LIN {X 0,Y 467.921,Z 515.715,A -85,B 0,C 180,E1 -7661.262,E2 -7661.262} C_VEL
LIN {X 0,Y 468.367,Z 505.748,A -85,B 0,C 180,E1 -7662.288,E2 -7662.288} C_VEL
LIN {X 0,Y 468.874,Z 494.586,A -85,B 0,C 180,E1 -7663.217,E2 -7663.217} C_VEL
LIN {X 0,Y 469.352,Z 483.029,A -85,B 0,C 180,E1 -7663.975,E2 -7663.975} C_VEL
LIN {X 0,Y 469.873,Z 469.859,A -85,B 0,C 180,E1 -7664.623,E2 -7664.623} C_VEL
LIN {X 0,Y 468.217,Z 456.623,A -85,B 0,C 180,E1 -7665.144,E2 -7665.144} C_VEL
LIN {X 0,Y 467.024,Z 448.323,A -85,B 0,C 180,E1 -7665.389,E2 -7665.389} C_VEL
LIN {X 0,Y 467.272,Z 438.89,A -85,B 0,C 180,E1 -7668.638,E2 -7668.638} C_VEL
LIN {X 0,Y 467.516,Z 429.097,A -85,B 0,C 180,E1 -7672.077,E2 -7672.077} C_VEL
LIN {X 0,Y 467.845,Z 420.214,A -85,B 0,C 180,E1 -7675.278,E2 -7675.278} C_VEL
LIN {X 0,Y 468.188,Z 412.234,A -85,B 0,C 180,E1 -7678.222,E2 -7678.222} C_VEL
LIN {X 0,Y 468.623,Z 404.282,A -85,B 0,C 180,E1 -7681.258,E2 -7681.258} C_VEL
LIN {X 0,Y 469.224,Z 395.561,A -85,B 0,C 180,E1 -7684.694,E2 -7684.694} C_VEL
LIN {X 0,Y 469.214,Z 392.362,A -85,B 0,C 180,E1 -7686.018,E2 -7686.018} C_VEL
LIN {X 0,Y 468.571,Z 387.882,A -85,B 0,C 180,E1 -7687.951,E2 -7687.951} C_VEL
LIN {X 0,Y 467.585,Z 382.244,A -85,B 0,C 180,E1 -7690.549,E2 -7690.549} C_VEL
LIN {X 0,Y 467.557,Z 382.244,A -85,B 0,C 180,E1 -7693.82,E2 -7693.82} C_VEL
LIN {X 0,Y 467.559,Z 382.245,A -85,B 0,C 180,E1 -7696.255,E2 -7696.255} C_VEL
LIN {X 0,Y 467.579,Z 382.244,A -85,B 0,C 180,E1 -7698.726,E2 -7698.726} C_VEL
LIN {X 0,Y 467.573,Z 382.242,A -85,B 0,C 180,E1 -7701.956,E2 -7701.956} C_VEL
LIN {X 0,Y 467.568,Z 382.246,A -85,B 0,C 180,E1 -7705.167,E2 -7705.167} C_VEL
LIN {X 0,Y 467.591,Z 382.241,A -85,B 0,C 180,E1 -7708.26,E2 -7708.26} C_VEL
LIN {X 0,Y 467.566,Z 382.244,A -85,B 0,C 180,E1 -7711.249,E2 -7711.249} C_VEL
LIN {X 0,Y 467.581,Z 382.24,A -85,B 0,C 180,E1 -7714.158,E2 -7714.158} C_VEL
LIN {X 0,Y 467.588,Z 382.242,A -85,B 0,C 180,E1 -7716.996,E2 -7716.996} C_VEL
LIN {X 0,Y 467.634,Z 382.236,A -85,B 0,C 180,E1 -7719.777,E2 -7719.777} C_VEL
LIN {X 0,Y 467.609,Z 382.238,A -85,B 0,C 180,E1 -7722.506,E2 -7722.506} C_VEL
LIN {X 0,Y 467.61,Z 382.24,A -85,B 0,C 180,E1 -7725.196,E2 -7725.196} C_VEL
LIN {X 0,Y 467.667,Z 382.231,A -85,B 0,C 180,E1 -7727.854,E2 -7727.854} C_VEL
LIN {X 0,Y 467.679,Z 382.23,A -85,B 0,C 180,E1 -7731.356,E2 -7731.356} C_VEL
LIN {X 0,Y 467.736,Z 382.221,A -85,B 0,C 180,E1 -7733.962,E2 -7733.962} C_VEL
LIN {X 0,Y 467.866,Z 382.208,A -85,B 0,C 180,E1 -7737.416,E2 -7737.416} C_VEL
LIN {X 0,Y 467.889,Z 382.203,A -85,B 0,C 180,E1 -7739.999,E2 -7739.999} C_VEL
LIN {X 0,Y 467.857,Z 382.208,A -85,B 0,C 180,E1 -7742.582,E2 -7742.582} C_VEL
LIN {X 0,Y 467.72,Z 382.224,A -85,B 0,C 180,E1 -7746.037,E2 -7746.037} C_VEL
LIN {X 0,Y 467.672,Z 382.231,A -85,B 0,C 180,E1 -7748.642,E2 -7748.642} C_VEL
LIN {X 0,Y 467.665,Z 382.232,A -85,B 0,C 180,E1 -7752.144,E2 -7752.144} C_VEL
LIN {X 0,Y 467.647,Z 382.232,A -85,B 0,C 180,E1 -7755.694,E2 -7755.694} C_VEL
LIN {X 0,Y 467.629,Z 382.235,A -85,B 0,C 180,E1 -7759.307,E2 -7759.307} C_VEL
LIN {X 0,Y 467.542,Z 382.247,A -85,B 0,C 180,E1 -7762.073,E2 -7762.073} C_VEL
LIN {X 0,Y 467.592,Z 382.241,A -85,B 0,C 180,E1 -7764.887,E2 -7764.887} C_VEL
LIN {X 0,Y 467.616,Z 382.235,A -85,B 0,C 180,E1 -7767.768,E2 -7767.768} C_VEL
LIN {X 0,Y 467.574,Z 382.244,A -85,B 0,C 180,E1 -7771.043,E2 -7771.043} C_VEL
LIN {X 0,Y 467.594,Z 382.241,A -85,B 0,C 180,E1 -7774.24,E2 -7774.24} C_VEL
LIN {X 0,Y 467.548,Z 382.246,A -85,B 0,C 180,E1 -7777.183,E2 -7777.183} C_VEL
LIN {X 0,Y 467.575,Z 382.244,A -85,B 0,C 180,E1 -7780.264,E2 -7780.264} C_VEL
LIN {X 0,Y 467.565,Z 382.244,A -85,B 0,C 180,E1 -7782.561,E2 -7782.561} C_VEL
LIN {X 0,Y 467.569,Z 382.243,A -85,B 0,C 180,E1 -7785.05,E2 -7785.05} C_VEL
LIN {X 0,Y 467.577,Z 382.244,A -85,B 0,C 180,E1 -7788.595,E2 -7788.595} C_VEL
LIN {X 0,Y 467.569,Z 382.243,A -85,B 0,C 180,E1 -7791.953,E2 -7791.953} C_VEL
LIN {X 0,Y 467.57,Z 382.243,A -85,B 0,C 180,E1 -7795.165,E2 -7795.165} C_VEL
LIN {X 0,Y 467.585,Z 382.242,A -85,B 0,C 180,E1 -7798.257,E2 -7798.257} C_VEL
LIN {X 0,Y 467.576,Z 382.241,A -85,B 0,C 180,E1 -7801.248,E2 -7801.248} C_VEL
LIN {X 0,Y 467.611,Z 382.239,A -85,B 0,C 180,E1 -7804.158,E2 -7804.158} C_VEL
LIN {X 0,Y 467.577,Z 382.243,A -85,B 0,C 180,E1 -7806.993,E2 -7806.993} C_VEL
LIN {X 0,Y 467.622,Z 382.237,A -85,B 0,C 180,E1 -7809.774,E2 -7809.774} C_VEL
LIN {X 0,Y 467.605,Z 382.242,A -85,B 0,C 180,E1 -7812.504,E2 -7812.504} C_VEL
LIN {X 0,Y 467.595,Z 382.239,A -85,B 0,C 180,E1 -7815.401,E2 -7815.401} C_VEL
LIN {X 0,Y 466.923,Z 382.325,A -85,B 0,C 180,E1 -7816.12,E2 -7816.12} C_VEL
LIN {X 0,Y 464.081,Z 382.675,A -85,B 0,C 180,E1 -7817.288,E2 -7817.288} C_VEL
LIN {X 0,Y 461.683,Z 382.978,A -85,B 0,C 180,E1 -7818.23,E2 -7818.23} C_VEL
LIN {X 0,Y 460.656,Z 383.105,A -85,B 0,C 180,E1 -7818.958,E2 -7818.958} C_VEL
LIN {X 0,Y 460.574,Z 383.113,A -85,B 0,C 180,E1 -7819.205,E2 -7819.205} C_VEL
LIN {X 0,Y 460.711,Z 383.098,A -85,B 0,C 180,E1 -7822.539,E2 -7822.539} C_VEL
LIN {X 0,Y 460.689,Z 383.1,A -85,B 0,C 180,E1 -7824.745,E2 -7824.745} C_VEL
LIN {X 0,Y 460.794,Z 383.087,A -85,B 0,C 180,E1 -7827.374,E2 -7827.374} C_VEL
LIN {X 0,Y 460.845,Z 383.083,A -85,B 0,C 180,E1 -7829.997,E2 -7829.997} C_VEL
LIN {X 0,Y 460.816,Z 383.086,A -85,B 0,C 180,E1 -7832.619,E2 -7832.619} C_VEL
LIN {X 0,Y 460.702,Z 383.099,A -85,B 0,C 180,E1 -7836.127,E2 -7836.127} C_VEL
LIN {X 0,Y 460.618,Z 383.109,A -85,B 0,C 180,E1 -7838.773,E2 -7838.773} C_VEL
LIN {X 0,Y 460.621,Z 383.109,A -85,B 0,C 180,E1 -7842.453,E2 -7842.453} C_VEL
LIN {X 0,Y 460.606,Z 383.113,A -85,B 0,C 180,E1 -7846.004,E2 -7846.004} C_VEL
LIN {X 0,Y 460.552,Z 383.117,A -85,B 0,C 180,E1 -7849.612,E2 -7849.612} C_VEL
LIN {X 0,Y 460.497,Z 383.126,A -85,B 0,C 180,E1 -7852.425,E2 -7852.425} C_VEL
LIN {X 0,Y 460.526,Z 383.12,A -85,B 0,C 180,E1 -7855.292,E2 -7855.292} C_VEL
LIN {X 0,Y 460.314,Z 383.15,A -85,B 0,C 180,E1 -7858.244,E2 -7858.244} C_VEL
LIN {X 0,Y 459.937,Z 383.378,A -85,B 0,C 180,E1 -7861.296,E2 -7861.296} C_VEL
LIN {X 0,Y 459.851,Z 386.637,A -85,B 0,C 180,E1 -7864.43,E2 -7864.43} C_VEL
LIN {X 0,Y 459.799,Z 390.069,A -85,B 0,C 180,E1 -7867.685,E2 -7867.685} C_VEL
LIN {X 0,Y 459.766,Z 392.69,A -85,B 0,C 180,E1 -7870.157,E2 -7870.157} C_VEL
LIN {X 0,Y 459.691,Z 396.273,A -85,B 0,C 180,E1 -7873.464,E2 -7873.464} C_VEL
LIN {X 0,Y 459.701,Z 399.614,A -85,B 0,C 180,E1 -7876.494,E2 -7876.494} C_VEL
LIN {X 0,Y 463.013,Z 414.025,A -85,B 0,C 180,E1 -7877.08,E2 -7877.08} C_VEL
LIN {X 0,Y 463.229,Z 419.464,A -85,B 0,C 180,E1 -7877.321,E2 -7877.321} C_VEL
LIN {X 0,Y 462.847,Z 431.199,A -85,B 0,C 180,E1 -7877.934,E2 -7877.934} C_VEL
LIN {X 0,Y 462.335,Z 443.116,A -85,B 0,C 180,E1 -7878.751,E2 -7878.751} C_VEL
LIN {X 0,Y 461.772,Z 454.579,A -85,B 0,C 180,E1 -7879.747,E2 -7879.747} C_VEL
LIN {X 0,Y 461.288,Z 464.913,A -85,B 0,C 180,E1 -7880.883,E2 -7880.883} C_VEL
LIN {X 0,Y 460.796,Z 474.093,A -85,B 0,C 180,E1 -7882.13,E2 -7882.13} C_VEL
LIN {X 0,Y 460.424,Z 482.007,A -85,B 0,C 180,E1 -7883.467,E2 -7883.467} C_VEL
LIN {X 0,Y 460.136,Z 488.259,A -85,B 0,C 180,E1 -7884.791,E2 -7884.791} C_VEL
LIN {X 0,Y 459.903,Z 493.202,A -85,B 0,C 180,E1 -7886.104,E2 -7886.104} C_VEL
LIN {X 0,Y 459.764,Z 497.612,A -85,B 0,C 180,E1 -7887.656,E2 -7887.656} C_VEL
LIN {X 0,Y 459.612,Z 500.119,A -85,B 0,C 180,E1 -7888.895,E2 -7888.895} C_VEL
LIN {X 0,Y 459.544,Z 502.273,A -85,B 0,C 180,E1 -7890.65,E2 -7890.65} C_VEL
LIN {X 0,Y 459.507,Z 502.75,A -85,B 0,C 180,E1 -7891.698,E2 -7891.698} C_VEL
LIN {X 0,Y 459.506,Z 502.726,A -85,B 0,C 180,E1 -7892.689,E2 -7892.689} C_VEL
LIN {X 0,Y 459.591,Z 501.374,A -85,B 0,C 180,E1 -7894.44,E2 -7894.44} C_VEL
LIN {X 0,Y 459.697,Z 499.578,A -85,B 0,C 180,E1 -7895.621,E2 -7895.621} C_VEL
LIN {X 0,Y 459.851,Z 496.301,A -85,B 0,C 180,E1 -7897.064,E2 -7897.064} C_VEL
LIN {X 0,Y 460.043,Z 491.012,A -85,B 0,C 180,E1 -7898.717,E2 -7898.717} C_VEL
LIN {X 0,Y 460.329,Z 484.96,A -85,B 0,C 180,E1 -7900.142,E2 -7900.142} C_VEL
LIN {X 0,Y 460.726,Z 477.332,A -85,B 0,C 180,E1 -7901.548,E2 -7901.548} C_VEL
LIN {X 0,Y 461.138,Z 469.536,A -85,B 0,C 180,E1 -7902.712,E2 -7902.712} C_VEL
LIN {X 0,Y 461.631,Z 459.665,A -85,B 0,C 180,E1 -7903.913,E2 -7903.913} C_VEL
LIN {X 0,Y 462.141,Z 449.461,A -85,B 0,C 180,E1 -7904.905,E2 -7904.905} C_VEL
LIN {X 0,Y 462.714,Z 437.651,A -85,B 0,C 180,E1 -7905.824,E2 -7905.824} C_VEL
LIN {X 0,Y 463.137,Z 426.76,A -85,B 0,C 180,E1 -7906.488,E2 -7906.488} C_VEL
LIN {X 0,Y 463.465,Z 416.28,A -85,B 0,C 180,E1 -7906.981,E2 -7906.981} C_VEL
LIN {X 0,Y 460.771,Z 404.535,A -85,B 0,C 180,E1 -7907.495,E2 -7907.495} C_VEL
LIN {X 0,Y 459.906,Z 400.872,A -85,B 0,C 180,E1 -7907.648,E2 -7907.648} C_VEL
LIN {X 0,Y 459.915,Z 397.286,A -85,B 0,C 180,E1 -7911.211,E2 -7911.211} C_VEL
LIN {X 0,Y 460.001,Z 394.662,A -85,B 0,C 180,E1 -7913.861,E2 -7913.861} C_VEL
LIN {X 0,Y 460.164,Z 392.942,A -85,B 0,C 180,E1 -7915.621,E2 -7915.621} C_VEL
LIN {X 0,Y 460.271,Z 389.556,A -85,B 0,C 180,E1 -7919.126,E2 -7919.126} C_VEL
LIN {X 0,Y 460.513,Z 387.881,A -85,B 0,C 180,E1 -7920.875,E2 -7920.875} C_VEL
LIN {X 0,Y 460.546,Z 383.831,A -85,B 0,C 180,E1 -7925.254,E2 -7925.254} C_VEL
LIN {X 0,Y 460.524,Z 383.125,A -85,B 0,C 180,E1 -7926.133,E2 -7926.133} C_VEL
LIN {X 0,Y 460.593,Z 383.116,A -85,B 0,C 180,E1 -7927.894,E2 -7927.894} C_VEL
LIN {X 0,Y 460.584,Z 383.116,A -85,B 0,C 180,E1 -7930.551,E2 -7930.551} C_VEL
LIN {X 0,Y 460.559,Z 383.119,A -85,B 0,C 180,E1 -7933.233,E2 -7933.233} C_VEL
LIN {X 0,Y 460.586,Z 383.114,A -85,B 0,C 180,E1 -7936.009,E2 -7936.009} C_VEL
LIN {X 0,Y 460.542,Z 383.12,A -85,B 0,C 180,E1 -7938.906,E2 -7938.906} C_VEL
LIN {X 0,Y 460.531,Z 383.119,A -85,B 0,C 180,E1 -7941.486,E2 -7941.486} C_VEL
LIN {X 0,Y 460.523,Z 383.119,A -85,B 0,C 180,E1 -7944.334,E2 -7944.334} C_VEL
LIN {X 0,Y 460.553,Z 383.117,A -85,B 0,C 180,E1 -7947.246,E2 -7947.246} C_VEL
LIN {X 0,Y 460.497,Z 383.124,A -85,B 0,C 180,E1 -7950.242,E2 -7950.242} C_VEL
LIN {X 0,Y 460.501,Z 383.124,A -85,B 0,C 180,E1 -7953.328,E2 -7953.328} C_VEL
LIN {X 0,Y 460.455,Z 383.13,A -85,B 0,C 180,E1 -7956.532,E2 -7956.532} C_VEL
LIN {X 0,Y 460.56,Z 383.118,A -85,B 0,C 180,E1 -7959.86,E2 -7959.86} C_VEL
LIN {X 0,Y 460.52,Z 383.125,A -85,B 0,C 180,E1 -7962.908,E2 -7962.908} C_VEL
LIN {X 0,Y 460.502,Z 383.126,A -85,B 0,C 180,E1 -7965.832,E2 -7965.832} C_VEL
LIN {X 0,Y 460.554,Z 383.166,A -85,B 0,C 180,E1 -7968.151,E2 -7968.151} C_VEL
LIN {X 0,Y 461.514,Z 388.734,A -85,B 0,C 180,E1 -7971.371,E2 -7971.371} C_VEL
LIN {X 0,Y 462.217,Z 393.26,A -85,B 0,C 180,E1 -7973.695,E2 -7973.695} C_VEL
LIN {X 0,Y 462.049,Z 397.702,A -85,B 0,C 180,E1 -7975.756,E2 -7975.756} C_VEL
LIN {X 0,Y 461.476,Z 404.849,A -85,B 0,C 180,E1 -7978.82,E2 -7978.82} C_VEL
LIN {X 0,Y 460.949,Z 413.207,A -85,B 0,C 180,E1 -7982.168,E2 -7982.168} C_VEL
LIN {X 0,Y 460.688,Z 419.887,A -85,B 0,C 180,E1 -7984.717,E2 -7984.717} C_VEL
LIN {X 0,Y 460.362,Z 428.911,A -85,B 0,C 180,E1 -7988.04,E2 -7988.04} C_VEL
LIN {X 0,Y 460.132,Z 436.905,A -85,B 0,C 180,E1 -7990.879,E2 -7990.879} C_VEL
LIN {X 0,Y 459.921,Z 446.946,A -85,B 0,C 180,E1 -7994.338,E2 -7994.338} C_VEL
LIN {X 0,Y 461.798,Z 460.563,A -85,B 0,C 180,E1 -7994.778,E2 -7994.778} C_VEL
LIN {X 0,Y 462.902,Z 471.743,A -85,B 0,C 180,E1 -7995.271,E2 -7995.271} C_VEL
LIN {X 0,Y 462.342,Z 483.982,A -85,B 0,C 180,E1 -7995.927,E2 -7995.927} C_VEL
LIN {X 0,Y 461.725,Z 496.525,A -85,B 0,C 180,E1 -7996.806,E2 -7996.806} C_VEL
LIN {X 0,Y 461.226,Z 506.53,A -85,B 0,C 180,E1 -7997.686,E2 -7997.686} C_VEL
LIN {X 0,Y 460.792,Z 516.676,A -85,B 0,C 180,E1 -7998.79,E2 -7998.79} C_VEL
LIN {X 0,Y 460.32,Z 526.54,A -85,B 0,C 180,E1 -8000.113,E2 -8000.113} C_VEL
LIN {X 0,Y 460.02,Z 534.432,A -85,B 0,C 180,E1 -8001.437,E2 -8001.437} C_VEL
LIN {X 0,Y 459.773,Z 541.699,A -85,B 0,C 180,E1 -8002.979,E2 -8002.979} C_VEL
LIN {X 0,Y 459.681,Z 546.549,A -85,B 0,C 180,E1 -8004.3,E2 -8004.3} C_VEL
LIN {X 0,Y 459.58,Z 550.258,A -85,B 0,C 180,E1 -8005.618,E2 -8005.618} C_VEL
LIN {X 0,Y 459.626,Z 552.182,A -85,B 0,C 180,E1 -8006.497,E2 -8006.497} C_VEL
LIN {X 0,Y 459.621,Z 553.624,A -85,B 0,C 180,E1 -8007.374,E2 -8007.374} C_VEL
LIN {X 0,Y 459.63,Z 554.658,A -85,B 0,C 180,E1 -8008.251,E2 -8008.251} C_VEL
LIN {X 0,Y 459.554,Z 555.294,A -85,B 0,C 180,E1 -8009.127,E2 -8009.127} C_VEL
LIN {X 0,Y 459.531,Z 555.527,A -85,B 0,C 180,E1 -8010.003,E2 -8010.003} C_VEL
LIN {X 0,Y 459.631,Z 554.72,A -85,B 0,C 180,E1 -8011.756,E2 -8011.756} C_VEL
LIN {X 0,Y 459.623,Z 553.72,A -85,B 0,C 180,E1 -8012.632,E2 -8012.632} C_VEL
LIN {X 0,Y 459.627,Z 552.303,A -85,B 0,C 180,E1 -8013.51,E2 -8013.51} C_VEL
LIN {X 0,Y 459.63,Z 549.329,A -85,B 0,C 180,E1 -8014.827,E2 -8014.827} C_VEL
LIN {X 0,Y 459.719,Z 544.241,A -85,B 0,C 180,E1 -8016.434,E2 -8016.434} C_VEL
LIN {X 0,Y 459.896,Z 538.06,A -85,B 0,C 180,E1 -8017.908,E2 -8017.908} C_VEL
LIN {X 0,Y 460.18,Z 531.048,A -85,B 0,C 180,E1 -8019.231,E2 -8019.231} C_VEL
LIN {X 0,Y 460.527,Z 522.257,A -85,B 0,C 180,E1 -8020.555,E2 -8020.555} C_VEL
LIN {X 0,Y 461.13,Z 512.301,A -85,B 0,C 180,E1 -8021.765,E2 -8021.765} C_VEL
LIN {X 0,Y 461.487,Z 502.127,A -85,B 0,C 180,E1 -8022.765,E2 -8022.765} C_VEL
LIN {X 0,Y 462.02,Z 491.009,A -85,B 0,C 180,E1 -8023.64,E2 -8023.64} C_VEL
LIN {X 0,Y 462.655,Z 478.556,A -85,B 0,C 180,E1 -8024.406,E2 -8024.406} C_VEL
LIN {X 0,Y 462.896,Z 469.283,A -85,B 0,C 180,E1 -8024.848,E2 -8024.848} C_VEL
LIN {X 0,Y 461.122,Z 455.923,A -85,B 0,C 180,E1 -8025.384,E2 -8025.384} C_VEL
LIN {X 0,Y 459.94,Z 447.939,A -85,B 0,C 180,E1 -8025.636,E2 -8025.636} C_VEL
LIN {X 0,Y 460.202,Z 439.025,A -85,B 0,C 180,E1 -8028.765,E2 -8028.765} C_VEL
LIN {X 0,Y 460.426,Z 430.104,A -85,B 0,C 180,E1 -8031.963,E2 -8031.963} C_VEL
LIN {X 0,Y 460.747,Z 422.328,A -85,B 0,C 180,E1 -8034.804,E2 -8034.804} C_VEL
LIN {X 0,Y 461.158,Z 413.292,A -85,B 0,C 180,E1 -8038.195,E2 -8038.195} C_VEL
LIN {X 0,Y 461.579,Z 405.572,A -85,B 0,C 180,E1 -8041.18,E2 -8041.18} C_VEL
LIN {X 0,Y 462.254,Z 396.524,A -85,B 0,C 180,E1 -8044.814,E2 -8044.814} C_VEL
LIN {X 0,Y 462.171,Z 392.819,A -85,B 0,C 180,E1 -8046.377,E2 -8046.377} C_VEL
LIN {X 0,Y 461.232,Z 386.951,A -85,B 0,C 180,E1 -8049.003,E2 -8049.003} C_VEL
LIN {X 0,Y 460.557,Z 383.119,A -85,B 0,C 180,E1 -8050.813,E2 -8050.813} C_VEL
LIN {X 0,Y 460.517,Z 383.121,A -85,B 0,C 180,E1 -8054.17,E2 -8054.17} C_VEL
LIN {X 0,Y 460.493,Z 383.126,A -85,B 0,C 180,E1 -8057.105,E2 -8057.105} C_VEL
LIN {X 0,Y 460.526,Z 383.12,A -85,B 0,C 180,E1 -8060.136,E2 -8060.136} C_VEL
LIN {X 0,Y 460.485,Z 383.127,A -85,B 0,C 180,E1 -8063.471,E2 -8063.471} C_VEL
LIN {X 0,Y 460.529,Z 383.121,A -85,B 0,C 180,E1 -8066.674,E2 -8066.674} C_VEL
LIN {X 0,Y 460.52,Z 383.12,A -85,B 0,C 180,E1 -8069.76,E2 -8069.76} C_VEL
LIN {X 0,Y 460.542,Z 383.119,A -85,B 0,C 180,E1 -8072.754,E2 -8072.754} C_VEL
LIN {X 0,Y 460.535,Z 383.121,A -85,B 0,C 180,E1 -8075.667,E2 -8075.667} C_VEL
LIN {X 0,Y 460.535,Z 383.119,A -85,B 0,C 180,E1 -8078.578,E2 -8078.578} C_VEL
LIN {X 0,Y 460.598,Z 383.114,A -85,B 0,C 180,E1 -8081.311,E2 -8081.311} C_VEL
LIN {X 0,Y 460.618,Z 383.109,A -85,B 0,C 180,E1 -8084.059,E2 -8084.059} C_VEL
LIN {X 0,Y 460.621,Z 383.109,A -85,B 0,C 180,E1 -8087.665,E2 -8087.665} C_VEL
LIN {X 0,Y 460.629,Z 383.108,A -85,B 0,C 180,E1 -8091.223,E2 -8091.223} C_VEL
LIN {X 0,Y 460.703,Z 383.097,A -85,B 0,C 180,E1 -8093.869,E2 -8093.869} C_VEL
LIN {X 0,Y 460.807,Z 383.087,A -85,B 0,C 180,E1 -8097.377,E2 -8097.377} C_VEL
LIN {X 0,Y 460.859,Z 383.079,A -85,B 0,C 180,E1 -8099.999,E2 -8099.999} C_VEL
LIN {X 0,Y 460.798,Z 383.088,A -85,B 0,C 180,E1 -8102.622,E2 -8102.622} C_VEL
LIN {X 0,Y 460.684,Z 383.1,A -85,B 0,C 180,E1 -8106.129,E2 -8106.129} C_VEL
LIN {X 0,Y 460.623,Z 383.109,A -85,B 0,C 180,E1 -8108.775,E2 -8108.775} C_VEL
LIN {X 0,Y 460.606,Z 383.113,A -85,B 0,C 180,E1 -8112.434,E2 -8112.434} C_VEL
LIN {X 0,Y 460.61,Z 383.109,A -85,B 0,C 180,E1 -8115.996,E2 -8115.996} C_VEL
LIN {X 0,Y 460.576,Z 383.113,A -85,B 0,C 180,E1 -8119.614,E2 -8119.614} C_VEL
LIN {X 0,Y 460.518,Z 383.122,A -85,B 0,C 180,E1 -8122.427,E2 -8122.427} C_VEL
LIN {X 0,Y 460.556,Z 383.117,A -85,B 0,C 180,E1 -8125.795,E2 -8125.795} C_VEL
LIN {X 0,Y 460.546,Z 383.118,A -85,B 0,C 180,E1 -8128.232,E2 -8128.232} C_VEL
LIN {X 0,Y 460.527,Z 383.119,A -85,B 0,C 180,E1 -8131.281,E2 -8131.281} C_VEL
LIN {X 0,Y 460.537,Z 383.12,A -85,B 0,C 180,E1 -8134.503,E2 -8134.503} C_VEL
LIN {X 0,Y 460.504,Z 383.123,A -85,B 0,C 180,E1 -8137.622,E2 -8137.622} C_VEL
LIN {X 0,Y 460.539,Z 383.12,A -85,B 0,C 180,E1 -8140.266,E2 -8140.266} C_VEL
LIN {X 0,Y 460.513,Z 383.121,A -85,B 0,C 180,E1 -8143.372,E2 -8143.372} C_VEL
LIN {X 0,Y 460.513,Z 383.123,A -85,B 0,C 180,E1 -8146.623,E2 -8146.623} C_VEL
LIN {X 0,Y 460.538,Z 383.119,A -85,B 0,C 180,E1 -8149.73,E2 -8149.73} C_VEL
LIN {X 0,Y 460.504,Z 383.126,A -85,B 0,C 180,E1 -8152.522,E2 -8152.522} C_VEL
LIN {X 0,Y 460.551,Z 383.117,A -85,B 0,C 180,E1 -8155.622,E2 -8155.622} C_VEL
LIN {X 0,Y 460.54,Z 383.12,A -85,B 0,C 180,E1 -8158.742,E2 -8158.742} C_VEL
LIN {X 0,Y 460.582,Z 383.115,A -85,B 0,C 180,E1 -8162.252,E2 -8162.252} C_VEL
LIN {X 0,Y 460.56,Z 383.117,A -85,B 0,C 180,E1 -8164.703,E2 -8164.703} C_VEL
LIN {X 0,Y 460.511,Z 383.123,A -85,B 0,C 180,E1 -8167.569,E2 -8167.569} C_VEL
LIN {X 0,Y 460.568,Z 383.116,A -85,B 0,C 180,E1 -8170.382,E2 -8170.382} C_VEL
LIN {X 0,Y 460.562,Z 383.114,A -85,B 0,C 180,E1 -8173.143,E2 -8173.143} C_VEL
LIN {X 0,Y 460.552,Z 383.118,A -85,B 0,C 180,E1 -8175.865,E2 -8175.865} C_VEL
LIN {X 0,Y 460.608,Z 383.111,A -85,B 0,C 180,E1 -8178.556,E2 -8178.556} C_VEL
LIN {X 0,Y 460.574,Z 383.113,A -85,B 0,C 180,E1 -8179.205,E2 -8179.205} C_VEL
LIN {X 0,Y 459.917,Z 383.198,A -85,B 0,C 180,E1 -8179.935,E2 -8179.935} C_VEL
LIN {X 0,Y 457.097,Z 383.552,A -85,B 0,C 180,E1 -8181.121,E2 -8181.121} C_VEL
LIN {X 0,Y 454.716,Z 383.847,A -85,B 0,C 180,E1 -8182.078,E2 -8182.078} C_VEL
LIN {X 0,Y 453.703,Z 383.971,A -85,B 0,C 180,E1 -8182.817,E2 -8182.817} C_VEL
LIN {X 0,Y 453.625,Z 383.98,A -85,B 0,C 180,E1 -8183.067,E2 -8183.067} C_VEL
LIN {X 0,Y 453.663,Z 383.976,A -85,B 0,C 180,E1 -8184.664,E2 -8184.664} C_VEL
LIN {X 0,Y 453.738,Z 383.966,A -85,B 0,C 180,E1 -8187.333,E2 -8187.333} C_VEL
LIN {X 0,Y 453.815,Z 383.959,A -85,B 0,C 180,E1 -8189.997,E2 -8189.997} C_VEL
LIN {X 0,Y 453.756,Z 383.964,A -85,B 0,C 180,E1 -8192.66,E2 -8192.66} C_VEL
LIN {X 0,Y 453.669,Z 383.976,A -85,B 0,C 180,E1 -8196.222,E2 -8196.222} C_VEL
LIN {X 0,Y 453.582,Z 383.985,A -85,B 0,C 180,E1 -8198.91,E2 -8198.91} C_VEL
LIN {X 0,Y 453.588,Z 383.984,A -85,B 0,C 180,E1 -8202.547,E2 -8202.547} C_VEL
LIN {X 0,Y 453.541,Z 383.992,A -85,B 0,C 180,E1 -8206.192,E2 -8206.192} C_VEL
LIN {X 0,Y 453.504,Z 383.995,A -85,B 0,C 180,E1 -8209.038,E2 -8209.038} C_VEL
LIN {X 0,Y 453.46,Z 384.002,A -85,B 0,C 180,E1 -8211.833,E2 -8211.833} C_VEL
LIN {X 0,Y 453.49,Z 383.995,A -85,B 0,C 180,E1 -8214.731,E2 -8214.731} C_VEL
LIN {X 0,Y 453.337,Z 384.018,A -85,B 0,C 180,E1 -8217.711,E2 -8217.711} C_VEL
LIN {X 0,Y 452.926,Z 384.075,A -85,B 0,C 180,E1 -8220.796,E2 -8220.796} C_VEL
LIN {X 0,Y 452.874,Z 384.19,A -85,B 0,C 180,E1 -8221.405,E2 -8221.405} C_VEL
LIN {X 0,Y 452.794,Z 387.534,A -85,B 0,C 180,E1 -8224.652,E2 -8224.652} C_VEL
LIN {X 0,Y 452.747,Z 390.692,A -85,B 0,C 180,E1 -8227.66,E2 -8227.66} C_VEL
LIN {X 0,Y 452.681,Z 393.925,A -85,B 0,C 180,E1 -8230.691,E2 -8230.691} C_VEL
LIN {X 0,Y 452.634,Z 397.827,A -85,B 0,C 180,E1 -8234.317,E2 -8234.317} C_VEL
LIN {X 0,Y 452.641,Z 399.971,A -85,B 0,C 180,E1 -8236.268,E2 -8236.268} C_VEL
LIN {X 0,Y 455.934,Z 414.289,A -85,B 0,C 180,E1 -8236.852,E2 -8236.852} C_VEL
LIN {X 0,Y 456.407,Z 418.655,A -85,B 0,C 180,E1 -8237.057,E2 -8237.057} C_VEL
LIN {X 0,Y 455.989,Z 431.188,A -85,B 0,C 180,E1 -8237.708,E2 -8237.708} C_VEL
LIN {X 0,Y 455.444,Z 443.242,A -85,B 0,C 180,E1 -8238.541,E2 -8238.541} C_VEL
LIN {X 0,Y 454.832,Z 454.602,A -85,B 0,C 180,E1 -8239.537,E2 -8239.537} C_VEL
LIN {X 0,Y 454.359,Z 464.73,A -85,B 0,C 180,E1 -8240.653,E2 -8240.653} C_VEL
LIN {X 0,Y 453.789,Z 474.492,A -85,B 0,C 180,E1 -8241.99,E2 -8241.99} C_VEL
LIN {X 0,Y 453.402,Z 482.206,A -85,B 0,C 180,E1 -8243.307,E2 -8243.307} C_VEL
LIN {X 0,Y 453.091,Z 488.725,A -85,B 0,C 180,E1 -8244.706,E2 -8244.706} C_VEL
LIN {X 0,Y 452.848,Z 493.644,A -85,B 0,C 180,E1 -8246.035,E2 -8246.035} C_VEL
LIN {X 0,Y 452.704,Z 498.061,A -85,B 0,C 180,E1 -8247.617,E2 -8247.617} C_VEL
LIN {X 0,Y 452.505,Z 501.043,A -85,B 0,C 180,E1 -8249.168,E2 -8249.168} C_VEL
LIN {X 0,Y 452.468,Z 502.495,A -85,B 0,C 180,E1 -8250.428,E2 -8250.428} C_VEL
LIN {X 0,Y 452.416,Z 503.013,A -85,B 0,C 180,E1 -8251.213,E2 -8251.213} C_VEL
LIN {X 0,Y 452.411,Z 503.197,A -85,B 0,C 180,E1 -8252.299,E2 -8252.299} C_VEL
LIN {X 0,Y 452.446,Z 502.892,A -85,B 0,C 180,E1 -8253.227,E2 -8253.227} C_VEL
LIN {X 0,Y 452.504,Z 502.069,A -85,B 0,C 180,E1 -8254.254,E2 -8254.254} C_VEL
LIN {X 0,Y 452.55,Z 500.783,A -85,B 0,C 180,E1 -8255.21,E2 -8255.21} C_VEL
LIN {X 0,Y 452.745,Z 497.722,A -85,B 0,C 180,E1 -8256.752,E2 -8256.752} C_VEL
LIN {X 0,Y 452.914,Z 493.826,A -85,B 0,C 180,E1 -8258.136,E2 -8258.136} C_VEL
LIN {X 0,Y 453.151,Z 488.507,A -85,B 0,C 180,E1 -8259.577,E2 -8259.577} C_VEL
LIN {X 0,Y 453.485,Z 481.699,A -85,B 0,C 180,E1 -8261.008,E2 -8261.008} C_VEL
LIN {X 0,Y 453.982,Z 473.16,A -85,B 0,C 180,E1 -8262.431,E2 -8262.431} C_VEL
LIN {X 0,Y 454.522,Z 464.332,A -85,B 0,C 180,E1 -8263.613,E2 -8263.613} C_VEL
LIN {X 0,Y 454.983,Z 454.695,A -85,B 0,C 180,E1 -8264.662,E2 -8264.662} C_VEL
LIN {X 0,Y 455.57,Z 444.076,A -85,B 0,C 180,E1 -8265.597,E2 -8265.597} C_VEL
LIN {X 0,Y 456.09,Z 432.537,A -85,B 0,C 180,E1 -8266.407,E2 -8266.407} C_VEL
LIN {X 0,Y 456.573,Z 419.658,A -85,B 0,C 180,E1 -8267.087,E2 -8267.087} C_VEL
LIN {X 0,Y 456.28,Z 415.433,A -85,B 0,C 180,E1 -8267.284,E2 -8267.284} C_VEL
LIN {X 0,Y 452.856,Z 401.356,A -85,B 0,C 180,E1 -8267.903,E2 -8267.903} C_VEL
LIN {X 0,Y 452.864,Z 398.185,A -85,B 0,C 180,E1 -8271.073,E2 -8271.073} C_VEL
LIN {X 0,Y 452.95,Z 395.562,A -85,B 0,C 180,E1 -8273.766,E2 -8273.766} C_VEL
LIN {X 0,Y 453.126,Z 393.81,A -85,B 0,C 180,E1 -8275.553,E2 -8275.553} C_VEL
LIN {X 0,Y 453.227,Z 390.435,A -85,B 0,C 180,E1 -8279.112,E2 -8279.112} C_VEL
LIN {X 0,Y 453.478,Z 388.773,A -85,B 0,C 180,E1 -8280.889,E2 -8280.889} C_VEL
LIN {X 0,Y 453.522,Z 384.723,A -85,B 0,C 180,E1 -8285.336,E2 -8285.336} C_VEL
LIN {X 0,Y 453.482,Z 384.003,A -85,B 0,C 180,E1 -8286.229,E2 -8286.229} C_VEL
LIN {X 0,Y 453.541,Z 383.994,A -85,B 0,C 180,E1 -8288.017,E2 -8288.017} C_VEL
LIN {X 0,Y 453.535,Z 383.993,A -85,B 0,C 180,E1 -8290.717,E2 -8290.717} C_VEL
LIN {X 0,Y 453.504,Z 383.998,A -85,B 0,C 180,E1 -8293.442,E2 -8293.442} C_VEL
LIN {X 0,Y 453.523,Z 383.996,A -85,B 0,C 180,E1 -8296.197,E2 -8296.197} C_VEL
LIN {X 0,Y 453.491,Z 383.999,A -85,B 0,C 180,E1 -8299.045,E2 -8299.045} C_VEL
LIN {X 0,Y 453.472,Z 383.999,A -85,B 0,C 180,E1 -8301.837,E2 -8301.837} C_VEL
LIN {X 0,Y 453.498,Z 383.995,A -85,B 0,C 180,E1 -8304.736,E2 -8304.736} C_VEL
LIN {X 0,Y 453.508,Z 383.995,A -85,B 0,C 180,E1 -8307.964,E2 -8307.964} C_VEL
LIN {X 0,Y 453.454,Z 384.002,A -85,B 0,C 180,E1 -8310.762,E2 -8310.762} C_VEL
LIN {X 0,Y 453.45,Z 384.003,A -85,B 0,C 180,E1 -8313.916,E2 -8313.916} C_VEL
LIN {X 0,Y 453.447,Z 384.003,A -85,B 0,C 180,E1 -8317.191,E2 -8317.191} C_VEL
LIN {X 0,Y 453.512,Z 383.996,A -85,B 0,C 180,E1 -8319.448,E2 -8319.448} C_VEL
LIN {X 0,Y 453.469,Z 384.003,A -85,B 0,C 180,E1 -8322.995,E2 -8322.995} C_VEL
LIN {X 0,Y 453.455,Z 384.003,A -85,B 0,C 180,E1 -8325.784,E2 -8325.784} C_VEL
LIN {X 0,Y 453.512,Z 384.041,A -85,B 0,C 180,E1 -8327.718,E2 -8327.718} C_VEL
LIN {X 0,Y 454.354,Z 388.949,A -85,B 0,C 180,E1 -8330.662,E2 -8330.662} C_VEL
LIN {X 0,Y 455.183,Z 394.03,A -85,B 0,C 180,E1 -8333.407,E2 -8333.407} C_VEL
LIN {X 0,Y 455.156,Z 397.71,A -85,B 0,C 180,E1 -8335.163,E2 -8335.163} C_VEL
LIN {X 0,Y 454.571,Z 404.727,A -85,B 0,C 180,E1 -8338.292,E2 -8338.292} C_VEL
LIN {X 0,Y 453.923,Z 413.613,A -85,B 0,C 180,E1 -8341.949,E2 -8341.949} C_VEL
LIN {X 0,Y 453.634,Z 420.872,A -85,B 0,C 180,E1 -8344.787,E2 -8344.787} C_VEL
LIN {X 0,Y 453.275,Z 429.888,A -85,B 0,C 180,E1 -8348.158,E2 -8348.158} C_VEL
LIN {X 0,Y 453.045,Z 438.125,A -85,B 0,C 180,E1 -8351.136,E2 -8351.136} C_VEL
LIN {X 0,Y 452.853,Z 446.636,A -85,B 0,C 180,E1 -8354.078,E2 -8354.078} C_VEL
LIN {X 0,Y 454.775,Z 459.997,A -85,B 0,C 180,E1 -8354.525,E2 -8354.525} C_VEL
LIN {X 0,Y 455.963,Z 472.582,A -85,B 0,C 180,E1 -8355.099,E2 -8355.099} C_VEL
LIN {X 0,Y 455.333,Z 485.389,A -85,B 0,C 180,E1 -8355.82,E2 -8355.82} C_VEL
LIN {X 0,Y 454.801,Z 496.155,A -85,B 0,C 180,E1 -8356.601,E2 -8356.601} C_VEL
LIN {X 0,Y 454.245,Z 506.142,A -85,B 0,C 180,E1 -8357.494,E2 -8357.494} C_VEL
LIN {X 0,Y 453.792,Z 516.278,A -85,B 0,C 180,E1 -8358.615,E2 -8358.615} C_VEL
LIN {X 0,Y 453.268,Z 526.122,A -85,B 0,C 180,E1 -8359.958,E2 -8359.958} C_VEL
LIN {X 0,Y 452.952,Z 534.004,A -85,B 0,C 180,E1 -8361.302,E2 -8361.302} C_VEL
LIN {X 0,Y 452.693,Z 541.267,A -85,B 0,C 180,E1 -8362.869,E2 -8362.869} C_VEL
LIN {X 0,Y 452.579,Z 546.123,A -85,B 0,C 180,E1 -8364.21,E2 -8364.21} C_VEL
LIN {X 0,Y 452.501,Z 549.841,A -85,B 0,C 180,E1 -8365.549,E2 -8365.549} C_VEL
LIN {X 0,Y 452.525,Z 551.766,A -85,B 0,C 180,E1 -8366.442,E2 -8366.442} C_VEL
LIN {X 0,Y 452.543,Z 553.212,A -85,B 0,C 180,E1 -8367.333,E2 -8367.333} C_VEL
LIN {X 0,Y 452.538,Z 554.25,A -85,B 0,C 180,E1 -8368.223,E2 -8368.223} C_VEL
LIN {X 0,Y 452.49,Z 554.888,A -85,B 0,C 180,E1 -8369.113,E2 -8369.113} C_VEL
LIN {X 0,Y 452.465,Z 555.121,A -85,B 0,C 180,E1 -8370.003,E2 -8370.003} C_VEL
LIN {X 0,Y 452.49,Z 554.913,A -85,B 0,C 180,E1 -8370.893,E2 -8370.893} C_VEL
LIN {X 0,Y 452.539,Z 554.311,A -85,B 0,C 180,E1 -8371.783,E2 -8371.783} C_VEL
LIN {X 0,Y 452.545,Z 553.311,A -85,B 0,C 180,E1 -8372.674,E2 -8372.674} C_VEL
LIN {X 0,Y 452.526,Z 551.888,A -85,B 0,C 180,E1 -8373.565,E2 -8373.565} C_VEL
LIN {X 0,Y 452.561,Z 548.911,A -85,B 0,C 180,E1 -8374.903,E2 -8374.903} C_VEL
LIN {X 0,Y 452.615,Z 544.309,A -85,B 0,C 180,E1 -8376.399,E2 -8376.399} C_VEL
LIN {X 0,Y 452.843,Z 537.624,A -85,B 0,C 180,E1 -8378.032,E2 -8378.032} C_VEL
LIN {X 0,Y 453.116,Z 530.596,A -85,B 0,C 180,E1 -8379.376,E2 -8379.376} C_VEL
LIN {X 0,Y 453.514,Z 521.793,A -85,B 0,C 180,E1 -8380.72,E2 -8380.72} C_VEL
LIN {X 0,Y 454.117,Z 511.821,A -85,B 0,C 180,E1 -8381.949,E2 -8381.949} C_VEL
LIN {X 0,Y 454.497,Z 501.621,A -85,B 0,C 180,E1 -8382.965,E2 -8382.965} C_VEL
LIN {X 0,Y 455.075,Z 490.489,A -85,B 0,C 180,E1 -8383.853,E2 -8383.853} C_VEL
LIN {X 0,Y 455.778,Z 478.015,A -85,B 0,C 180,E1 -8384.628,E2 -8384.628} C_VEL
LIN {X 0,Y 455.93,Z 469.98,A -85,B 0,C 180,E1 -8385.023,E2 -8385.023} C_VEL
LIN {X 0,Y 454.204,Z 456.5,A -85,B 0,C 180,E1 -8385.585,E2 -8385.585} C_VEL
LIN {X 0,Y 452.896,Z 447.599,A -85,B 0,C 180,E1 -8385.875,E2 -8385.875} C_VEL
LIN {X 0,Y 453.121,Z 438.857,A -85,B 0,C 180,E1 -8389.012,E2 -8389.012} C_VEL
LIN {X 0,Y 453.4,Z 429.781,A -85,B 0,C 180,E1 -8392.322,E2 -8392.322} C_VEL
LIN {X 0,Y 453.736,Z 422.048,A -85,B 0,C 180,E1 -8395.214,E2 -8395.214} C_VEL
LIN {X 0,Y 454.186,Z 413.034,A -85,B 0,C 180,E1 -8398.668,E2 -8398.668} C_VEL
LIN {X 0,Y 454.655,Z 405.211,A -85,B 0,C 180,E1 -8401.768,E2 -8401.768} C_VEL
LIN {X 0,Y 455.241,Z 397.682,A -85,B 0,C 180,E1 -8404.837,E2 -8404.837} C_VEL
LIN {X 0,Y 455.131,Z 393.64,A -85,B 0,C 180,E1 -8406.585,E2 -8406.585} C_VEL
LIN {X 0,Y 453.93,Z 386.239,A -85,B 0,C 180,E1 -8409.983,E2 -8409.983} C_VEL
LIN {X 0,Y 453.501,Z 383.998,A -85,B 0,C 180,E1 -8411.124,E2 -8411.124} C_VEL
LIN {X 0,Y 453.494,Z 383.997,A -85,B 0,C 180,E1 -8414.529,E2 -8414.529} C_VEL
LIN {X 0,Y 453.462,Z 384,A -85,B 0,C 180,E1 -8418.07,E2 -8418.07} C_VEL
LIN {X 0,Y 453.46,Z 384.001,A -85,B 0,C 180,E1 -8420.802,E2 -8420.802} C_VEL
LIN {X 0,Y 453.463,Z 384,A -85,B 0,C 180,E1 -8423.917,E2 -8423.917} C_VEL
LIN {X 0,Y 453.487,Z 383.998,A -85,B 0,C 180,E1 -8427.151,E2 -8427.151} C_VEL
LIN {X 0,Y 453.479,Z 383.997,A -85,B 0,C 180,E1 -8430.268,E2 -8430.268} C_VEL
LIN {X 0,Y 453.476,Z 384.001,A -85,B 0,C 180,E1 -8433.291,E2 -8433.291} C_VEL
LIN {X 0,Y 453.506,Z 383.995,A -85,B 0,C 180,E1 -8436.238,E2 -8436.238} C_VEL
LIN {X 0,Y 453.495,Z 383.997,A -85,B 0,C 180,E1 -8439.118,E2 -8439.118} C_VEL
LIN {X 0,Y 453.515,Z 383.992,A -85,B 0,C 180,E1 -8441.944,E2 -8441.944} C_VEL
LIN {X 0,Y 453.548,Z 383.99,A -85,B 0,C 180,E1 -8444.726,E2 -8444.726} C_VEL
LIN {X 0,Y 453.568,Z 383.988,A -85,B 0,C 180,E1 -8448.378,E2 -8448.378} C_VEL
LIN {X 0,Y 453.595,Z 383.985,A -85,B 0,C 180,E1 -8451.086,E2 -8451.086} C_VEL
LIN {X 0,Y 453.67,Z 383.973,A -85,B 0,C 180,E1 -8453.774,E2 -8453.774} C_VEL
LIN {X 0,Y 453.751,Z 383.966,A -85,B 0,C 180,E1 -8457.336,E2 -8457.336} C_VEL
LIN {X 0,Y 453.829,Z 383.954,A -85,B 0,C 180,E1 -8459.999,E2 -8459.999} C_VEL
LIN {X 0,Y 453.742,Z 383.967,A -85,B 0,C 180,E1 -8462.663,E2 -8462.663} C_VEL
LIN {X 0,Y 453.651,Z 383.976,A -85,B 0,C 180,E1 -8466.225,E2 -8466.225} C_VEL
LIN {X 0,Y 453.59,Z 383.985,A -85,B 0,C 180,E1 -8468.913,E2 -8468.913} C_VEL
LIN {X 0,Y 453.574,Z 383.988,A -85,B 0,C 180,E1 -8472.528,E2 -8472.528} C_VEL
LIN {X 0,Y 453.554,Z 383.989,A -85,B 0,C 180,E1 -8476.195,E2 -8476.195} C_VEL
LIN {X 0,Y 453.526,Z 383.993,A -85,B 0,C 180,E1 -8479.038,E2 -8479.038} C_VEL
LIN {X 0,Y 453.485,Z 383.997,A -85,B 0,C 180,E1 -8481.835,E2 -8481.835} C_VEL
LIN {X 0,Y 453.507,Z 383.996,A -85,B 0,C 180,E1 -8484.734,E2 -8484.734} C_VEL
LIN {X 0,Y 453.531,Z 383.99,A -85,B 0,C 180,E1 -8487.956,E2 -8487.956} C_VEL
LIN {X 0,Y 453.472,Z 383.997,A -85,B 0,C 180,E1 -8491.523,E2 -8491.523} C_VEL
LIN {X 0,Y 453.493,Z 383.999,A -85,B 0,C 180,E1 -8494.775,E2 -8494.775} C_VEL
LIN {X 0,Y 453.463,Z 384.001,A -85,B 0,C 180,E1 -8498.31,E2 -8498.31} C_VEL
LIN {X 0,Y 453.499,Z 383.998,A -85,B 0,C 180,E1 -8500.607,E2 -8500.607} C_VEL
LIN {X 0,Y 453.464,Z 384.001,A -85,B 0,C 180,E1 -8504.22,E2 -8504.22} C_VEL
LIN {X 0,Y 453.453,Z 384.003,A -85,B 0,C 180,E1 -8507.001,E2 -8507.001} C_VEL
LIN {X 0,Y 453.498,Z 383.995,A -85,B 0,C 180,E1 -8509.407,E2 -8509.407} C_VEL
LIN {X 0,Y 453.456,Z 384.001,A -85,B 0,C 180,E1 -8512.808,E2 -8512.808} C_VEL
LIN {X 0,Y 453.481,Z 383.998,A -85,B 0,C 180,E1 -8516.085,E2 -8516.085} C_VEL
LIN {X 0,Y 453.478,Z 383.998,A -85,B 0,C 180,E1 -8519.238,E2 -8519.238} C_VEL
LIN {X 0,Y 453.537,Z 383.992,A -85,B 0,C 180,E1 -8522.295,E2 -8522.295} C_VEL
LIN {X 0,Y 453.515,Z 383.992,A -85,B 0,C 180,E1 -8525.263,E2 -8525.263} C_VEL
LIN {X 0,Y 453.48,Z 384.001,A -85,B 0,C 180,E1 -8528.412,E2 -8528.412} C_VEL
LIN {X 0,Y 453.521,Z 383.994,A -85,B 0,C 180,E1 -8531.006,E2 -8531.006} C_VEL
LIN {X 0,Y 453.567,Z 383.988,A -85,B 0,C 180,E1 -8533.877,E2 -8533.877} C_VEL
LIN {X 0,Y 453.561,Z 383.986,A -85,B 0,C 180,E1 -8537.468,E2 -8537.468} C_VEL
LIN {X 0,Y 453.588,Z 383.983,A -85,B 0,C 180,E1 -8541.084,E2 -8541.084} C_VEL
LIN {X 0,Y 453.625,Z 383.98,A -85,B 0,C 180,E1 -8543.067,E2 -8543.067} C_VEL
LIN {X 0,Y 452.939,Z 384.066,A -85,B 0,C 180,E1 -8543.808,E2 -8543.808} C_VEL
LIN {X 0,Y 449.992,Z 384.431,A -85,B 0,C 180,E1 -8545.01,E2 -8545.01} C_VEL
LIN {X 0,Y 447.567,Z 384.737,A -85,B 0,C 180,E1 -8545.979,E2 -8545.979} C_VEL
LIN {X 0,Y 446.623,Z 384.853,A -85,B 0,C 180,E1 -8546.729,E2 -8546.729} C_VEL
LIN {X 0,Y 446.598,Z 384.854,A -85,B 0,C 180,E1 -8546.983,E2 -8546.983} C_VEL
LIN {X 0,Y 446.785,Z 384.834,A -85,B 0,C 180,E1 -8549.997,E2 -8549.997} C_VEL
LIN {X 0,Y 446.7,Z 384.843,A -85,B 0,C 180,E1 -8552.702,E2 -8552.702} C_VEL
LIN {X 0,Y 446.638,Z 384.852,A -85,B 0,C 180,E1 -8556.32,E2 -8556.32} C_VEL
LIN {X 0,Y 446.528,Z 384.863,A -85,B 0,C 180,E1 -8559.052,E2 -8559.052} C_VEL
LIN {X 0,Y 446.52,Z 384.864,A -85,B 0,C 180,E1 -8562.726,E2 -8562.726} C_VEL
LIN {X 0,Y 446.48,Z 384.87,A -85,B 0,C 180,E1 -8566.455,E2 -8566.455} C_VEL
LIN {X 0,Y 446.452,Z 384.873,A -85,B 0,C 180,E1 -8569.3,E2 -8569.3} C_VEL
LIN {X 0,Y 446.402,Z 384.881,A -85,B 0,C 180,E1 -8572.196,E2 -8572.196} C_VEL
LIN {X 0,Y 446.427,Z 384.875,A -85,B 0,C 180,E1 -8575.15,E2 -8575.15} C_VEL
LIN {X 0,Y 446.233,Z 384.904,A -85,B 0,C 180,E1 -8578.191,E2 -8578.191} C_VEL
LIN {X 0,Y 445.842,Z 384.957,A -85,B 0,C 180,E1 -8581.34,E2 -8581.34} C_VEL
LIN {X 0,Y 445.734,Z 388.154,A -85,B 0,C 180,E1 -8584.579,E2 -8584.579} C_VEL
LIN {X 0,Y 445.651,Z 391.667,A -85,B 0,C 180,E1 -8587.955,E2 -8587.955} C_VEL
LIN {X 0,Y 445.625,Z 394.677,A -85,B 0,C 180,E1 -8590.8,E2 -8590.8} C_VEL
LIN {X 0,Y 445.538,Z 398.064,A -85,B 0,C 180,E1 -8593.946,E2 -8593.946} C_VEL
LIN {X 0,Y 445.599,Z 400.514,A -85,B 0,C 180,E1 -8596.04,E2 -8596.04} C_VEL
LIN {X 0,Y 448.792,Z 414.199,A -85,B 0,C 180,E1 -8596.605,E2 -8596.605} C_VEL
LIN {X 0,Y 449.545,Z 419.114,A -85,B 0,C 180,E1 -8596.845,E2 -8596.845} C_VEL
LIN {X 0,Y 449.094,Z 431.724,A -85,B 0,C 180,E1 -8597.513,E2 -8597.513} C_VEL
LIN {X 0,Y 448.589,Z 442.428,A -85,B 0,C 180,E1 -8598.254,E2 -8598.254} C_VEL
LIN {X 0,Y 447.956,Z 453.653,A -85,B 0,C 180,E1 -8599.232,E2 -8599.232} C_VEL
LIN {X 0,Y 447.444,Z 463.661,A -85,B 0,C 180,E1 -8600.314,E2 -8600.314} C_VEL
LIN {X 0,Y 446.965,Z 472.498,A -85,B 0,C 180,E1 -8601.49,E2 -8601.49} C_VEL
LIN {X 0,Y 446.496,Z 479.955,A -85,B 0,C 180,E1 -8602.7,E2 -8602.7} C_VEL
LIN {X 0,Y 446.135,Z 486.991,A -85,B 0,C 180,E1 -8604.111,E2 -8604.111} C_VEL
LIN {X 0,Y 445.884,Z 492.248,A -85,B 0,C 180,E1 -8605.43,E2 -8605.43} C_VEL
LIN {X 0,Y 445.665,Z 497.424,A -85,B 0,C 180,E1 -8607.128,E2 -8607.128} C_VEL
LIN {X 0,Y 445.473,Z 500.61,A -85,B 0,C 180,E1 -8608.627,E2 -8608.627} C_VEL
LIN {X 0,Y 445.375,Z 502.707,A -85,B 0,C 180,E1 -8610.205,E2 -8610.205} C_VEL
LIN {X 0,Y 445.344,Z 503.637,A -85,B 0,C 180,E1 -8612.086,E2 -8612.086} C_VEL
LIN {X 0,Y 445.391,Z 502.951,A -85,B 0,C 180,E1 -8613.781,E2 -8613.781} C_VEL
LIN {X 0,Y 445.435,Z 501.902,A -85,B 0,C 180,E1 -8614.787,E2 -8614.787} C_VEL
LIN {X 0,Y 445.595,Z 499.621,A -85,B 0,C 180,E1 -8616.163,E2 -8616.163} C_VEL
LIN {X 0,Y 445.801,Z 495.709,A -85,B 0,C 180,E1 -8617.769,E2 -8617.769} C_VEL
LIN {X 0,Y 446.026,Z 490.778,A -85,B 0,C 180,E1 -8619.236,E2 -8619.236} C_VEL
LIN {X 0,Y 446.394,Z 483.804,A -85,B 0,C 180,E1 -8620.83,E2 -8620.83} C_VEL
LIN {X 0,Y 446.853,Z 476.549,A -85,B 0,C 180,E1 -8622.141,E2 -8622.141} C_VEL
LIN {X 0,Y 447.363,Z 468.078,A -85,B 0,C 180,E1 -8623.378,E2 -8623.378} C_VEL
LIN {X 0,Y 447.946,Z 458.364,A -85,B 0,C 180,E1 -8624.532,E2 -8624.532} C_VEL
LIN {X 0,Y 448.554,Z 447.418,A -85,B 0,C 180,E1 -8625.583,E2 -8625.583} C_VEL
LIN {X 0,Y 449.109,Z 436.303,A -85,B 0,C 180,E1 -8626.425,E2 -8626.425} C_VEL
LIN {X 0,Y 449.648,Z 423.785,A -85,B 0,C 180,E1 -8627.16,E2 -8627.16} C_VEL
LIN {X 0,Y 449.66,Z 417.502,A -85,B 0,C 180,E1 -8627.464,E2 -8627.464} C_VEL
LIN {X 0,Y 446.56,Z 404.842,A -85,B 0,C 180,E1 -8628.054,E2 -8628.054} C_VEL
LIN {X 0,Y 445.786,Z 401.834,A -85,B 0,C 180,E1 -8628.174,E2 -8628.174} C_VEL
LIN {X 0,Y 445.837,Z 398.233,A -85,B 0,C 180,E1 -8631.845,E2 -8631.845} C_VEL
LIN {X 0,Y 446.089,Z 394.714,A -85,B 0,C 180,E1 -8635.483,E2 -8635.483} C_VEL
LIN {X 0,Y 446.184,Z 391.353,A -85,B 0,C 180,E1 -8639.098,E2 -8639.098} C_VEL
LIN {X 0,Y 446.444,Z 389.66,A -85,B 0,C 180,E1 -8640.903,E2 -8640.903} C_VEL
LIN {X 0,Y 446.498,Z 385.642,A -85,B 0,C 180,E1 -8645.42,E2 -8645.42} C_VEL
LIN {X 0,Y 446.445,Z 384.88,A -85,B 0,C 180,E1 -8646.327,E2 -8646.327} C_VEL
LIN {X 0,Y 446.52,Z 384.869,A -85,B 0,C 180,E1 -8648.144,E2 -8648.144} C_VEL
LIN {X 0,Y 446.487,Z 384.87,A -85,B 0,C 180,E1 -8650.889,E2 -8650.889} C_VEL
LIN {X 0,Y 446.453,Z 384.875,A -85,B 0,C 180,E1 -8653.659,E2 -8653.659} C_VEL
LIN {X 0,Y 446.466,Z 384.873,A -85,B 0,C 180,E1 -8656.461,E2 -8656.461} C_VEL
LIN {X 0,Y 446.438,Z 384.878,A -85,B 0,C 180,E1 -8659.305,E2 -8659.305} C_VEL
LIN {X 0,Y 446.411,Z 384.881,A -85,B 0,C 180,E1 -8662.201,E2 -8662.201} C_VEL
LIN {X 0,Y 446.443,Z 384.877,A -85,B 0,C 180,E1 -8665.154,E2 -8665.154} C_VEL
LIN {X 0,Y 446.454,Z 384.875,A -85,B 0,C 180,E1 -8668.181,E2 -8668.181} C_VEL
LIN {X 0,Y 446.39,Z 384.882,A -85,B 0,C 180,E1 -8671.303,E2 -8671.303} C_VEL
LIN {X 0,Y 446.403,Z 384.881,A -85,B 0,C 180,E1 -8674.526,E2 -8674.526} C_VEL
LIN {X 0,Y 446.415,Z 384.88,A -85,B 0,C 180,E1 -8678.087,E2 -8678.087} C_VEL
LIN {X 0,Y 446.424,Z 384.88,A -85,B 0,C 180,E1 -8680.924,E2 -8680.924} C_VEL
LIN {X 0,Y 446.423,Z 384.879,A -85,B 0,C 180,E1 -8683.844,E2 -8683.844} C_VEL
LIN {X 0,Y 446.446,Z 384.897,A -85,B 0,C 180,E1 -8687.25,E2 -8687.25} C_VEL
LIN {X 0,Y 447.31,Z 389.812,A -85,B 0,C 180,E1 -8690.343,E2 -8690.343} C_VEL
LIN {X 0,Y 448.238,Z 395.473,A -85,B 0,C 180,E1 -8693.435,E2 -8693.435} C_VEL
LIN {X 0,Y 448.106,Z 399.974,A -85,B 0,C 180,E1 -8695.63,E2 -8695.63} C_VEL
LIN {X 0,Y 447.441,Z 407.038,A -85,B 0,C 180,E1 -8698.784,E2 -8698.784} C_VEL
LIN {X 0,Y 446.848,Z 415.599,A -85,B 0,C 180,E1 -8702.361,E2 -8702.361} C_VEL
LIN {X 0,Y 446.482,Z 423.185,A -85,B 0,C 180,E1 -8705.351,E2 -8705.351} C_VEL
LIN {X 0,Y 446.208,Z 430.995,A -85,B 0,C 180,E1 -8708.324,E2 -8708.324} C_VEL
LIN {X 0,Y 445.972,Z 438.238,A -85,B 0,C 180,E1 -8711.003,E2 -8711.003} C_VEL
LIN {X 0,Y 445.78,Z 446.031,A -85,B 0,C 180,E1 -8713.792,E2 -8713.792} C_VEL
LIN {X 0,Y 447.686,Z 458.963,A -85,B 0,C 180,E1 -8714.238,E2 -8714.238} C_VEL
LIN {X 0,Y 449.088,Z 472.305,A -85,B 0,C 180,E1 -8714.866,E2 -8714.866} C_VEL
LIN {X 0,Y 448.42,Z 485.041,A -85,B 0,C 180,E1 -8715.597,E2 -8715.597} C_VEL
LIN {X 0,Y 447.785,Z 497.036,A -85,B 0,C 180,E1 -8716.494,E2 -8716.494} C_VEL
LIN {X 0,Y 447.152,Z 507.922,A -85,B 0,C 180,E1 -8717.523,E2 -8717.523} C_VEL
LIN {X 0,Y 446.699,Z 517.691,A -85,B 0,C 180,E1 -8718.662,E2 -8718.662} C_VEL
LIN {X 0,Y 446.212,Z 525.724,A -85,B 0,C 180,E1 -8719.797,E2 -8719.797} C_VEL
LIN {X 0,Y 445.872,Z 533.601,A -85,B 0,C 180,E1 -8721.163,E2 -8721.163} C_VEL
LIN {X 0,Y 445.615,Z 540.867,A -85,B 0,C 180,E1 -8722.755,E2 -8722.755} C_VEL
LIN {X 0,Y 445.492,Z 545.114,A -85,B 0,C 180,E1 -8723.931,E2 -8723.931} C_VEL
LIN {X 0,Y 445.426,Z 549.434,A -85,B 0,C 180,E1 -8725.479,E2 -8725.479} C_VEL
LIN {X 0,Y 445.425,Z 551.358,A -85,B 0,C 180,E1 -8726.385,E2 -8726.385} C_VEL
LIN {X 0,Y 445.467,Z 552.805,A -85,B 0,C 180,E1 -8727.291,E2 -8727.291} C_VEL
LIN {X 0,Y 445.451,Z 553.843,A -85,B 0,C 180,E1 -8728.195,E2 -8728.195} C_VEL
LIN {X 0,Y 445.427,Z 554.483,A -85,B 0,C 180,E1 -8729.099,E2 -8729.099} C_VEL
LIN {X 0,Y 445.401,Z 554.714,A -85,B 0,C 180,E1 -8730.003,E2 -8730.003} C_VEL
LIN {X 0,Y 445.428,Z 554.507,A -85,B 0,C 180,E1 -8730.907,E2 -8730.907} C_VEL
LIN {X 0,Y 445.452,Z 553.903,A -85,B 0,C 180,E1 -8731.811,E2 -8731.811} C_VEL
LIN {X 0,Y 445.468,Z 552.902,A -85,B 0,C 180,E1 -8732.716,E2 -8732.716} C_VEL
LIN {X 0,Y 445.426,Z 551.474,A -85,B 0,C 180,E1 -8733.622,E2 -8733.622} C_VEL
LIN {X 0,Y 445.492,Z 548.493,A -85,B 0,C 180,E1 -8734.981,E2 -8734.981} C_VEL
LIN {X 0,Y 445.561,Z 542.977,A -85,B 0,C 180,E1 -8736.752,E2 -8736.752} C_VEL
LIN {X 0,Y 445.77,Z 537.178,A -85,B 0,C 180,E1 -8738.161,E2 -8738.161} C_VEL
LIN {X 0,Y 446.059,Z 530.127,A -85,B 0,C 180,E1 -8739.526,E2 -8739.526} C_VEL
LIN {X 0,Y 446.513,Z 521.299,A -85,B 0,C 180,E1 -8740.89,E2 -8740.89} C_VEL
LIN {X 0,Y 447.11,Z 511.296,A -85,B 0,C 180,E1 -8742.139,E2 -8742.139} C_VEL
LIN {X 0,Y 447.538,Z 500.875,A -85,B 0,C 180,E1 -8743.185,E2 -8743.185} C_VEL
LIN {X 0,Y 448.176,Z 489.866,A -85,B 0,C 180,E1 -8744.07,E2 -8744.07} C_VEL
LIN {X 0,Y 448.756,Z 479.291,A -85,B 0,C 180,E1 -8744.746,E2 -8744.746} C_VEL
LIN {X 0,Y 448.939,Z 470.469,A -85,B 0,C 180,E1 -8745.205,E2 -8745.205} C_VEL
LIN {X 0,Y 447.226,Z 456.759,A -85,B 0,C 180,E1 -8745.795,E2 -8745.795} C_VEL
LIN {X 0,Y 445.833,Z 447.286,A -85,B 0,C 180,E1 -8746.108,E2 -8746.108} C_VEL
LIN {X 0,Y 446.112,Z 437.199,A -85,B 0,C 180,E1 -8749.801,E2 -8749.801} C_VEL
LIN {X 0,Y 446.454,Z 428.192,A -85,B 0,C 180,E1 -8753.178,E2 -8753.178} C_VEL
LIN {X 0,Y 446.807,Z 420.074,A -85,B 0,C 180,E1 -8756.287,E2 -8756.287} C_VEL
LIN {X 0,Y 447.297,Z 411.496,A -85,B 0,C 180,E1 -8759.668,E2 -8759.668} C_VEL
LIN {X 0,Y 447.796,Z 403.832,A -85,B 0,C 180,E1 -8762.786,E2 -8762.786} C_VEL
LIN {X 0,Y 448.276,Z 397.475,A -85,B 0,C 180,E1 -8765.459,E2 -8765.459} C_VEL
LIN {X 0,Y 448.08,Z 394.263,A -85,B 0,C 180,E1 -8766.877,E2 -8766.877} C_VEL
LIN {X 0,Y 446.919,Z 387.28,A -85,B 0,C 180,E1 -8770.149,E2 -8770.149} C_VEL
LIN {X 0,Y 446.436,Z 384.878,A -85,B 0,C 180,E1 -8771.393,E2 -8771.393} C_VEL
LIN {X 0,Y 446.435,Z 384.874,A -85,B 0,C 180,E1 -8775.109,E2 -8775.109} C_VEL
LIN {X 0,Y 446.42,Z 384.879,A -85,B 0,C 180,E1 -8778.607,E2 -8778.607} C_VEL
LIN {X 0,Y 446.423,Z 384.876,A -85,B 0,C 180,E1 -8781.923,E2 -8781.923} C_VEL
LIN {X 0,Y 446.435,Z 384.876,A -85,B 0,C 180,E1 -8785.477,E2 -8785.477} C_VEL
LIN {X 0,Y 446.427,Z 384.877,A -85,B 0,C 180,E1 -8788.7,E2 -8788.7} C_VEL
LIN {X 0,Y 446.462,Z 384.873,A -85,B 0,C 180,E1 -8791.83,E2 -8791.83} C_VEL
LIN {X 0,Y 446.446,Z 384.877,A -85,B 0,C 180,E1 -8794.846,E2 -8794.846} C_VEL
LIN {X 0,Y 446.462,Z 384.87,A -85,B 0,C 180,E1 -8798.245,E2 -8798.245} C_VEL
LIN {X 0,Y 446.464,Z 384.871,A -85,B 0,C 180,E1 -8801.649,E2 -8801.649} C_VEL
LIN {X 0,Y 446.518,Z 384.867,A -85,B 0,C 180,E1 -8804.479,E2 -8804.479} C_VEL
LIN {X 0,Y 446.528,Z 384.864,A -85,B 0,C 180,E1 -8808.193,E2 -8808.193} C_VEL
LIN {X 0,Y 446.542,Z 384.865,A -85,B 0,C 180,E1 -8810.944,E2 -8810.944} C_VEL
LIN {X 0,Y 446.64,Z 384.849,A -85,B 0,C 180,E1 -8813.675,E2 -8813.675} C_VEL
LIN {X 0,Y 446.698,Z 384.845,A -85,B 0,C 180,E1 -8817.294,E2 -8817.294} C_VEL
LIN {X 0,Y 446.799,Z 384.83,A -85,B 0,C 180,E1 -8819.999,E2 -8819.999} C_VEL
LIN {X 0,Y 446.689,Z 384.846,A -85,B 0,C 180,E1 -8822.705,E2 -8822.705} C_VEL
LIN {X 0,Y 446.62,Z 384.852,A -85,B 0,C 180,E1 -8826.323,E2 -8826.323} C_VEL
LIN {X 0,Y 446.538,Z 384.864,A -85,B 0,C 180,E1 -8829.054,E2 -8829.054} C_VEL
LIN {X 0,Y 446.532,Z 384.865,A -85,B 0,C 180,E1 -8832.729,E2 -8832.729} C_VEL
LIN {X 0,Y 446.498,Z 384.87,A -85,B 0,C 180,E1 -8836.458,E2 -8836.458} C_VEL
LIN {X 0,Y 446.477,Z 384.869,A -85,B 0,C 180,E1 -8839.302,E2 -8839.302} C_VEL
LIN {X 0,Y 446.426,Z 384.877,A -85,B 0,C 180,E1 -8842.198,E2 -8842.198} C_VEL
LIN {X 0,Y 446.449,Z 384.875,A -85,B 0,C 180,E1 -8845.152,E2 -8845.152} C_VEL
LIN {X 0,Y 446.493,Z 384.868,A -85,B 0,C 180,E1 -8848.177,E2 -8848.177} C_VEL
LIN {X 0,Y 446.425,Z 384.875,A -85,B 0,C 180,E1 -8851.773,E2 -8851.773} C_VEL
LIN {X 0,Y 446.435,Z 384.877,A -85,B 0,C 180,E1 -8854.521,E2 -8854.521} C_VEL
LIN {X 0,Y 446.416,Z 384.88,A -85,B 0,C 180,E1 -8858.076,E2 -8858.076} C_VEL
LIN {X 0,Y 446.424,Z 384.877,A -85,B 0,C 180,E1 -8861.39,E2 -8861.39} C_VEL
LIN {X 0,Y 446.455,Z 384.873,A -85,B 0,C 180,E1 -8865.102,E2 -8865.102} C_VEL
LIN {X 0,Y 446.422,Z 384.879,A -85,B 0,C 180,E1 -8868.606,E2 -8868.606} C_VEL
LIN {X 0,Y 446.428,Z 384.878,A -85,B 0,C 180,E1 -8870.969,E2 -8870.969} C_VEL
LIN {X 0,Y 446.424,Z 384.878,A -85,B 0,C 180,E1 -8874.372,E2 -8874.372} C_VEL
LIN {X 0,Y 446.425,Z 384.876,A -85,B 0,C 180,E1 -8877.636,E2 -8877.636} C_VEL
LIN {X 0,Y 446.449,Z 384.874,A -85,B 0,C 180,E1 -8880.788,E2 -8880.788} C_VEL
LIN {X 0,Y 446.479,Z 384.87,A -85,B 0,C 180,E1 -8883.846,E2 -8883.846} C_VEL
LIN {X 0,Y 446.43,Z 384.878,A -85,B 0,C 180,E1 -8886.821,E2 -8886.821} C_VEL
LIN {X 0,Y 446.444,Z 384.874,A -85,B 0,C 180,E1 -8889.734,E2 -8889.734} C_VEL
LIN {X 0,Y 446.461,Z 384.874,A -85,B 0,C 180,E1 -8892.594,E2 -8892.594} C_VEL
LIN {X 0,Y 446.468,Z 384.871,A -85,B 0,C 180,E1 -8895.409,E2 -8895.409} C_VEL
LIN {X 0,Y 446.515,Z 384.868,A -85,B 0,C 180,E1 -8898.19,E2 -8898.19} C_VEL
LIN {X 0,Y 446.596,Z 384.856,A -85,B 0,C 180,E1 -8901.855,E2 -8901.855} C_VEL
LIN {X 0,Y 446.637,Z 384.852,A -85,B 0,C 180,E1 -8904.579,E2 -8904.579} C_VEL
LIN {X 0,Y 446.598,Z 384.854,A -85,B 0,C 180,E1 -8906.983,E2 -8906.983} C_VEL
LIN {X 0,Y 446.074,Z 384.922,A -85,B 0,C 180,E1 -8907.736,E2 -8907.736} C_VEL
LIN {X 0,Y 443.265,Z 385.274,A -85,B 0,C 180,E1 -8908.959,E2 -8908.959} C_VEL
LIN {X 0,Y 440.792,Z 385.582,A -85,B 0,C 180,E1 -8909.946,E2 -8909.946} C_VEL
LIN {X 0,Y 439.709,Z 385.714,A -85,B 0,C 180,E1 -8910.71,E2 -8910.71} C_VEL
LIN {X 0,Y 439.615,Z 385.725,A -85,B 0,C 180,E1 -8910.968,E2 -8910.968} C_VEL
LIN {X 0,Y 439.647,Z 385.721,A -85,B 0,C 180,E1 -8912.745,E2 -8912.745} C_VEL
LIN {X 0,Y 439.609,Z 385.728,A -85,B 0,C 180,E1 -8916.422,E2 -8916.422} C_VEL
LIN {X 0,Y 439.49,Z 385.74,A -85,B 0,C 180,E1 -8919.198,E2 -8919.198} C_VEL
LIN {X 0,Y 439.49,Z 385.74,A -85,B 0,C 180,E1 -8922.723,E2 -8922.723} C_VEL
LIN {X 0,Y 439.445,Z 385.747,A -85,B 0,C 180,E1 -8926.351,E2 -8926.351} C_VEL
LIN {X 0,Y 439.385,Z 385.754,A -85,B 0,C 180,E1 -8929.623,E2 -8929.623} C_VEL
LIN {X 0,Y 439.348,Z 385.759,A -85,B 0,C 180,E1 -8932.572,E2 -8932.572} C_VEL
LIN {X 0,Y 439.36,Z 385.758,A -85,B 0,C 180,E1 -8935.583,E2 -8935.583} C_VEL
LIN {X 0,Y 439.126,Z 385.787,A -85,B 0,C 180,E1 -8938.689,E2 -8938.689} C_VEL
LIN {X 0,Y 438.826,Z 385.83,A -85,B 0,C 180,E1 -8940.825,E2 -8940.825} C_VEL
LIN {X 0,Y 438.719,Z 386.13,A -85,B 0,C 180,E1 -8941.908,E2 -8941.908} C_VEL
LIN {X 0,Y 438.637,Z 389.511,A -85,B 0,C 180,E1 -8945.221,E2 -8945.221} C_VEL
LIN {X 0,Y 438.573,Z 392.665,A -85,B 0,C 180,E1 -8948.262,E2 -8948.262} C_VEL
LIN {X 0,Y 438.535,Z 395.678,A -85,B 0,C 180,E1 -8951.131,E2 -8951.131} C_VEL
LIN {X 0,Y 438.46,Z 399.651,A -85,B 0,C 180,E1 -8954.845,E2 -8954.845} C_VEL
LIN {X 0,Y 438.498,Z 400.673,A -85,B 0,C 180,E1 -8955.779,E2 -8955.779} C_VEL
LIN {X 0,Y 441.709,Z 414.568,A -85,B 0,C 180,E1 -8956.37,E2 -8956.37} C_VEL
LIN {X 0,Y 442.633,Z 418.844,A -85,B 0,C 180,E1 -8956.591,E2 -8956.591} C_VEL
LIN {X 0,Y 442.228,Z 431.774,A -85,B 0,C 180,E1 -8957.283,E2 -8957.283} C_VEL
LIN {X 0,Y 441.663,Z 442.909,A -85,B 0,C 180,E1 -8958.063,E2 -8958.063} C_VEL
LIN {X 0,Y 441.01,Z 454.211,A -85,B 0,C 180,E1 -8959.066,E2 -8959.066} C_VEL
LIN {X 0,Y 440.468,Z 464.039,A -85,B 0,C 180,E1 -8960.147,E2 -8960.147} C_VEL
LIN {X 0,Y 440.027,Z 471.782,A -85,B 0,C 180,E1 -8961.18,E2 -8961.18} C_VEL
LIN {X 0,Y 439.48,Z 480.389,A -85,B 0,C 180,E1 -8962.579,E2 -8962.579} C_VEL
LIN {X 0,Y 439.107,Z 487.247,A -85,B 0,C 180,E1 -8963.973,E2 -8963.973} C_VEL
LIN {X 0,Y 438.842,Z 492.68,A -85,B 0,C 180,E1 -8965.354,E2 -8965.354} C_VEL
LIN {X 0,Y 438.597,Z 497.632,A -85,B 0,C 180,E1 -8966.99,E2 -8966.99} C_VEL
LIN {X 0,Y 438.479,Z 500.195,A -85,B 0,C 180,E1 -8968.147,E2 -8968.147} C_VEL
LIN {X 0,Y 438.337,Z 501.887,A -85,B 0,C 180,E1 -8969.133,E2 -8969.133} C_VEL
LIN {X 0,Y 438.288,Z 503.114,A -85,B 0,C 180,E1 -8970.194,E2 -8970.194} C_VEL
LIN {X 0,Y 438.258,Z 504.011,A -85,B 0,C 180,E1 -8971.873,E2 -8971.873} C_VEL
LIN {X 0,Y 438.312,Z 503.322,A -85,B 0,C 180,E1 -8973.874,E2 -8973.874} C_VEL
LIN {X 0,Y 438.407,Z 501.568,A -85,B 0,C 180,E1 -8975.368,E2 -8975.368} C_VEL
LIN {X 0,Y 438.628,Z 498.646,A -85,B 0,C 180,E1 -8976.887,E2 -8976.887} C_VEL
LIN {X 0,Y 438.82,Z 494.568,A -85,B 0,C 180,E1 -8978.386,E2 -8978.386} C_VEL
LIN {X 0,Y 439.109,Z 489.213,A -85,B 0,C 180,E1 -8979.874,E2 -8979.874} C_VEL
LIN {X 0,Y 439.513,Z 482.372,A -85,B 0,C 180,E1 -8981.35,E2 -8981.35} C_VEL
LIN {X 0,Y 439.989,Z 475.206,A -85,B 0,C 180,E1 -8982.598,E2 -8982.598} C_VEL
LIN {X 0,Y 440.555,Z 466.863,A -85,B 0,C 180,E1 -8983.79,E2 -8983.79} C_VEL
LIN {X 0,Y 441.116,Z 457.613,A -85,B 0,C 180,E1 -8984.878,E2 -8984.878} C_VEL
LIN {X 0,Y 441.725,Z 447.578,A -85,B 0,C 180,E1 -8985.837,E2 -8985.837} C_VEL
LIN {X 0,Y 442.297,Z 436.577,A -85,B 0,C 180,E1 -8986.68,E2 -8986.68} C_VEL
LIN {X 0,Y 442.837,Z 424.498,A -85,B 0,C 180,E1 -8987.402,E2 -8987.402} C_VEL
LIN {X 0,Y 442.872,Z 418.85,A -85,B 0,C 180,E1 -8987.682,E2 -8987.682} C_VEL
LIN {X 0,Y 439.764,Z 406.209,A -85,B 0,C 180,E1 -8988.302,E2 -8988.302} C_VEL
LIN {X 0,Y 438.718,Z 402.297,A -85,B 0,C 180,E1 -8988.479,E2 -8988.479} C_VEL
LIN {X 0,Y 438.769,Z 399.158,A -85,B 0,C 180,E1 -8991.712,E2 -8991.712} C_VEL
LIN {X 0,Y 438.97,Z 396.511,A -85,B 0,C 180,E1 -8994.488,E2 -8994.488} C_VEL
LIN {X 0,Y 438.905,Z 394.803,A -85,B 0,C 180,E1 -8996.329,E2 -8996.329} C_VEL
LIN {X 0,Y 439.14,Z 392.259,A -85,B 0,C 180,E1 -8999.084,E2 -8999.084} C_VEL
LIN {X 0,Y 439.41,Z 390.564,A -85,B 0,C 180,E1 -9000.917,E2 -9000.917} C_VEL
LIN {X 0,Y 439.474,Z 386.565,A -85,B 0,C 180,E1 -9005.507,E2 -9005.507} C_VEL
LIN {X 0,Y 439.412,Z 385.796,A -85,B 0,C 180,E1 -9006.429,E2 -9006.429} C_VEL
LIN {X 0,Y 439.485,Z 385.746,A -85,B 0,C 180,E1 -9008.276,E2 -9008.276} C_VEL
LIN {X 0,Y 439.439,Z 385.748,A -85,B 0,C 180,E1 -9011.065,E2 -9011.065} C_VEL
LIN {X 0,Y 439.404,Z 385.752,A -85,B 0,C 180,E1 -9013.882,E2 -9013.882} C_VEL
LIN {X 0,Y 439.429,Z 385.748,A -85,B 0,C 180,E1 -9016.732,E2 -9016.732} C_VEL
LIN {X 0,Y 439.402,Z 385.753,A -85,B 0,C 180,E1 -9019.627,E2 -9019.627} C_VEL
LIN {X 0,Y 439.353,Z 385.757,A -85,B 0,C 180,E1 -9022.577,E2 -9022.577} C_VEL
LIN {X 0,Y 439.384,Z 385.754,A -85,B 0,C 180,E1 -9025.587,E2 -9025.587} C_VEL
LIN {X 0,Y 439.395,Z 385.753,A -85,B 0,C 180,E1 -9028.676,E2 -9028.676} C_VEL
LIN {X 0,Y 439.345,Z 385.759,A -85,B 0,C 180,E1 -9031.863,E2 -9031.863} C_VEL
LIN {X 0,Y 439.374,Z 385.757,A -85,B 0,C 180,E1 -9035.159,E2 -9035.159} C_VEL
LIN {X 0,Y 439.376,Z 385.756,A -85,B 0,C 180,E1 -9038.596,E2 -9038.596} C_VEL
LIN {X 0,Y 439.381,Z 385.756,A -85,B 0,C 180,E1 -9041.263,E2 -9041.263} C_VEL
LIN {X 0,Y 439.388,Z 385.756,A -85,B 0,C 180,E1 -9044.732,E2 -9044.732} C_VEL
LIN {X 0,Y 439.406,Z 385.792,A -85,B 0,C 180,E1 -9046.775,E2 -9046.775} C_VEL
LIN {X 0,Y 440.373,Z 391.312,A -85,B 0,C 180,E1 -9050.336,E2 -9050.336} C_VEL
LIN {X 0,Y 441.245,Z 396.656,A -85,B 0,C 180,E1 -9053.361,E2 -9053.361} C_VEL
LIN {X 0,Y 441.213,Z 399.96,A -85,B 0,C 180,E1 -9055.015,E2 -9055.015} C_VEL
LIN {X 0,Y 440.517,Z 406.926,A -85,B 0,C 180,E1 -9058.237,E2 -9058.237} C_VEL
LIN {X 0,Y 439.908,Z 414.46,A -85,B 0,C 180,E1 -9061.485,E2 -9061.485} C_VEL
LIN {X 0,Y 439.581,Z 421.662,A -85,B 0,C 180,E1 -9064.431,E2 -9064.431} C_VEL
LIN {X 0,Y 439.237,Z 429.27,A -85,B 0,C 180,E1 -9067.422,E2 -9067.422} C_VEL
LIN {X 0,Y 438.964,Z 437.022,A -85,B 0,C 180,E1 -9070.358,E2 -9070.358} C_VEL
LIN {X 0,Y 438.736,Z 445.521,A -85,B 0,C 180,E1 -9073.5,E2 -9073.5} C_VEL
LIN {X 0,Y 440.81,Z 459.396,A -85,B 0,C 180,E1 -9073.996,E2 -9073.996} C_VEL
LIN {X 0,Y 442.173,Z 473.307,A -85,B 0,C 180,E1 -9074.682,E2 -9074.682} C_VEL
LIN {X 0,Y 441.536,Z 484.836,A -85,B 0,C 180,E1 -9075.368,E2 -9075.368} C_VEL
LIN {X 0,Y 440.864,Z 496.65,A -85,B 0,C 180,E1 -9076.27,E2 -9076.27} C_VEL
LIN {X 0,Y 440.179,Z 507.564,A -85,B 0,C 180,E1 -9077.322,E2 -9077.322} C_VEL
LIN {X 0,Y 439.694,Z 517.297,A -85,B 0,C 180,E1 -9078.479,E2 -9078.479} C_VEL
LIN {X 0,Y 439.187,Z 525.327,A -85,B 0,C 180,E1 -9079.633,E2 -9079.633} C_VEL
LIN {X 0,Y 438.814,Z 533.199,A -85,B 0,C 180,E1 -9081.02,E2 -9081.02} C_VEL
LIN {X 0,Y 438.537,Z 540.47,A -85,B 0,C 180,E1 -9082.638,E2 -9082.638} C_VEL
LIN {X 0,Y 438.392,Z 545.154,A -85,B 0,C 180,E1 -9083.97,E2 -9083.97} C_VEL
LIN {X 0,Y 438.355,Z 549.038,A -85,B 0,C 180,E1 -9085.406,E2 -9085.406} C_VEL
LIN {X 0,Y 438.327,Z 550.957,A -85,B 0,C 180,E1 -9086.326,E2 -9086.326} C_VEL
LIN {X 0,Y 438.392,Z 552.403,A -85,B 0,C 180,E1 -9087.247,E2 -9087.247} C_VEL
LIN {X 0,Y 438.366,Z 553.439,A -85,B 0,C 180,E1 -9088.166,E2 -9088.166} C_VEL
LIN {X 0,Y 438.366,Z 554.08,A -85,B 0,C 180,E1 -9089.085,E2 -9089.085} C_VEL
LIN {X 0,Y 438.339,Z 554.305,A -85,B 0,C 180,E1 -9090.003,E2 -9090.003} C_VEL
LIN {X 0,Y 438.367,Z 554.093,A -85,B 0,C 180,E1 -9090.922,E2 -9090.922} C_VEL
LIN {X 0,Y 438.367,Z 553.484,A -85,B 0,C 180,E1 -9091.841,E2 -9091.841} C_VEL
LIN {X 0,Y 438.393,Z 552.479,A -85,B 0,C 180,E1 -9092.76,E2 -9092.76} C_VEL
LIN {X 0,Y 438.33,Z 551.038,A -85,B 0,C 180,E1 -9093.68,E2 -9093.68} C_VEL
LIN {X 0,Y 438.422,Z 548.047,A -85,B 0,C 180,E1 -9095.061,E2 -9095.061} C_VEL
LIN {X 0,Y 438.453,Z 543.979,A -85,B 0,C 180,E1 -9096.446,E2 -9096.446} C_VEL
LIN {X 0,Y 438.672,Z 537.714,A -85,B 0,C 180,E1 -9098.062,E2 -9098.062} C_VEL
LIN {X 0,Y 438.964,Z 530.887,A -85,B 0,C 180,E1 -9099.448,E2 -9099.448} C_VEL
LIN {X 0,Y 439.382,Z 522.397,A -85,B 0,C 180,E1 -9100.836,E2 -9100.836} C_VEL
LIN {X 0,Y 439.947,Z 513.669,A -85,B 0,C 180,E1 -9101.989,E2 -9101.989} C_VEL
LIN {X 0,Y 440.459,Z 502.458,A -85,B 0,C 180,E1 -9103.194,E2 -9103.194} C_VEL
LIN {X 0,Y 441.163,Z 490.776,A -85,B 0,C 180,E1 -9104.181,E2 -9104.181} C_VEL
LIN {X 0,Y 441.86,Z 478.577,A -85,B 0,C 180,E1 -9104.982,E2 -9104.982} C_VEL
LIN {X 0,Y 441.944,Z 470.929,A -85,B 0,C 180,E1 -9105.392,E2 -9105.392} C_VEL
LIN {X 0,Y 440.263,Z 457.189,A -85,B 0,C 180,E1 -9106.005,E2 -9106.005} C_VEL
LIN {X 0,Y 438.764,Z 446.943,A -85,B 0,C 180,E1 -9106.355,E2 -9106.355} C_VEL
LIN {X 0,Y 439.014,Z 438.141,A -85,B 0,C 180,E1 -9109.647,E2 -9109.647} C_VEL
LIN {X 0,Y 439.374,Z 429.139,A -85,B 0,C 180,E1 -9113.075,E2 -9113.075} C_VEL
LIN {X 0,Y 439.812,Z 420.167,A -85,B 0,C 180,E1 -9116.582,E2 -9116.582} C_VEL
LIN {X 0,Y 440.317,Z 411.478,A -85,B 0,C 180,E1 -9120.079,E2 -9120.079} C_VEL
LIN {X 0,Y 440.797,Z 404.854,A -85,B 0,C 180,E1 -9122.829,E2 -9122.829} C_VEL
LIN {X 0,Y 441.269,Z 399.778,A -85,B 0,C 180,E1 -9124.988,E2 -9124.988} C_VEL
LIN {X 0,Y 441.156,Z 396.059,A -85,B 0,C 180,E1 -9126.635,E2 -9126.635} C_VEL
LIN {X 0,Y 440.033,Z 389.097,A -85,B 0,C 180,E1 -9129.947,E2 -9129.947} C_VEL
LIN {X 0,Y 439.389,Z 385.756,A -85,B 0,C 180,E1 -9131.699,E2 -9131.699} C_VEL
LIN {X 0,Y 439.389,Z 385.752,A -85,B 0,C 180,E1 -9135.268,E2 -9135.268} C_VEL
LIN {X 0,Y 439.381,Z 385.756,A -85,B 0,C 180,E1 -9138.747,E2 -9138.747} C_VEL
LIN {X 0,Y 439.377,Z 385.755,A -85,B 0,C 180,E1 -9141.61,E2 -9141.61} C_VEL
LIN {X 0,Y 439.408,Z 385.751,A -85,B 0,C 180,E1 -9144.844,E2 -9144.844} C_VEL
LIN {X 0,Y 439.382,Z 385.754,A -85,B 0,C 180,E1 -9148.14,E2 -9148.14} C_VEL
LIN {X 0,Y 439.417,Z 385.751,A -85,B 0,C 180,E1 -9151.606,E2 -9151.606} C_VEL
LIN {X 0,Y 439.385,Z 385.753,A -85,B 0,C 180,E1 -9154.413,E2 -9154.413} C_VEL
LIN {X 0,Y 439.376,Z 385.756,A -85,B 0,C 180,E1 -9157.424,E2 -9157.424} C_VEL
LIN {X 0,Y 439.454,Z 385.746,A -85,B 0,C 180,E1 -9160.663,E2 -9160.663} C_VEL
LIN {X 0,Y 439.474,Z 385.743,A -85,B 0,C 180,E1 -9164.224,E2 -9164.224} C_VEL
LIN {X 0,Y 439.495,Z 385.74,A -85,B 0,C 180,E1 -9168.001,E2 -9168.001} C_VEL
LIN {X 0,Y 439.516,Z 385.737,A -85,B 0,C 180,E1 -9171.725,E2 -9171.725} C_VEL
LIN {X 0,Y 439.621,Z 385.724,A -85,B 0,C 180,E1 -9174.495,E2 -9174.495} C_VEL
LIN {X 0,Y 439.643,Z 385.721,A -85,B 0,C 180,E1 -9178.167,E2 -9178.167} C_VEL
LIN {X 0,Y 439.768,Z 385.705,A -85,B 0,C 180,E1 -9179.999,E2 -9179.999} C_VEL
LIN {X 0,Y 439.639,Z 385.724,A -85,B 0,C 180,E1 -9182.748,E2 -9182.748} C_VEL
LIN {X 0,Y 439.572,Z 385.73,A -85,B 0,C 180,E1 -9186.425,E2 -9186.425} C_VEL
LIN {X 0,Y 439.502,Z 385.741,A -85,B 0,C 180,E1 -9189.201,E2 -9189.201} C_VEL
LIN {X 0,Y 439.476,Z 385.743,A -85,B 0,C 180,E1 -9192.936,E2 -9192.936} C_VEL
LIN {X 0,Y 439.456,Z 385.746,A -85,B 0,C 180,E1 -9196.346,E2 -9196.346} C_VEL
LIN {X 0,Y 439.411,Z 385.749,A -85,B 0,C 180,E1 -9199.625,E2 -9199.625} C_VEL
LIN {X 0,Y 439.372,Z 385.757,A -85,B 0,C 180,E1 -9202.574,E2 -9202.574} C_VEL
LIN {X 0,Y 439.396,Z 385.752,A -85,B 0,C 180,E1 -9205.584,E2 -9205.584} C_VEL
LIN {X 0,Y 439.422,Z 385.751,A -85,B 0,C 180,E1 -9208.672,E2 -9208.672} C_VEL
LIN {X 0,Y 439.376,Z 385.754,A -85,B 0,C 180,E1 -9212.028,E2 -9212.028} C_VEL
LIN {X 0,Y 439.399,Z 385.751,A -85,B 0,C 180,E1 -9215.338,E2 -9215.338} C_VEL
LIN {X 0,Y 439.374,Z 385.756,A -85,B 0,C 180,E1 -9218.595,E2 -9218.595} C_VEL
LIN {X 0,Y 439.387,Z 385.754,A -85,B 0,C 180,E1 -9221.253,E2 -9221.253} C_VEL
LIN {X 0,Y 439.403,Z 385.753,A -85,B 0,C 180,E1 -9224.728,E2 -9224.728} C_VEL
LIN {X 0,Y 439.388,Z 385.752,A -85,B 0,C 180,E1 -9227.792,E2 -9227.792} C_VEL
LIN {X 0,Y 439.393,Z 385.754,A -85,B 0,C 180,E1 -9230.221,E2 -9230.221} C_VEL
LIN {X 0,Y 439.378,Z 385.754,A -85,B 0,C 180,E1 -9233.71,E2 -9233.71} C_VEL
LIN {X 0,Y 439.375,Z 385.754,A -85,B 0,C 180,E1 -9237.051,E2 -9237.051} C_VEL
LIN {X 0,Y 439.384,Z 385.755,A -85,B 0,C 180,E1 -9240.271,E2 -9240.271} C_VEL
LIN {X 0,Y 439.43,Z 385.748,A -85,B 0,C 180,E1 -9243.393,E2 -9243.393} C_VEL
LIN {X 0,Y 439.388,Z 385.754,A -85,B 0,C 180,E1 -9246.427,E2 -9246.427} C_VEL
LIN {X 0,Y 439.388,Z 385.752,A -85,B 0,C 180,E1 -9249.394,E2 -9249.394} C_VEL
LIN {X 0,Y 439.429,Z 385.75,A -85,B 0,C 180,E1 -9252.307,E2 -9252.307} C_VEL
LIN {X 0,Y 439.445,Z 385.746,A -85,B 0,C 180,E1 -9255.171,E2 -9255.171} C_VEL
LIN {X 0,Y 439.481,Z 385.744,A -85,B 0,C 180,E1 -9257.998,E2 -9257.998} C_VEL
LIN {X 0,Y 439.544,Z 385.733,A -85,B 0,C 180,E1 -9261.723,E2 -9261.723} C_VEL
LIN {X 0,Y 439.612,Z 385.728,A -85,B 0,C 180,E1 -9264.492,E2 -9264.492} C_VEL
LIN {X 0,Y 439.629,Z 385.725,A -85,B 0,C 180,E1 -9268.165,E2 -9268.165} C_VEL
LIN {X 0,Y 439.755,Z 385.71,A -85,B 0,C 180,E1 -9269.997,E2 -9269.997} C_VEL
LIN {X 0,Y 439.615,Z 385.725,A -85,B 0,C 180,E1 -9270.968,E2 -9270.968} C_VEL
LIN {X 0,Y 438.898,Z 385.816,A -85,B 0,C 180,E1 -9271.733,E2 -9271.733} C_VEL
LIN {X 0,Y 435.916,Z 386.185,A -85,B 0,C 180,E1 -9272.972,E2 -9272.972} C_VEL
LIN {X 0,Y 433.463,Z 386.493,A -85,B 0,C 180,E1 -9273.972,E2 -9273.972} C_VEL
LIN {X 0,Y 432.489,Z 386.613,A -85,B 0,C 180,E1 -9274.746,E2 -9274.746} C_VEL
LIN {X 0,Y 432.452,Z 386.616,A -85,B 0,C 180,E1 -9275.008,E2 -9275.008} C_VEL
LIN {X 0,Y 432.575,Z 386.602,A -85,B 0,C 180,E1 -9277.676,E2 -9277.676} C_VEL
LIN {X 0,Y 432.397,Z 386.623,A -85,B 0,C 180,E1 -9281.243,E2 -9281.243} C_VEL
LIN {X 0,Y 432.371,Z 386.629,A -85,B 0,C 180,E1 -9284.108,E2 -9284.108} C_VEL
LIN {X 0,Y 432.383,Z 386.625,A -85,B 0,C 180,E1 -9287.008,E2 -9287.008} C_VEL
LIN {X 0,Y 432.322,Z 386.636,A -85,B 0,C 180,E1 -9289.957,E2 -9289.957} C_VEL
LIN {X 0,Y 432.302,Z 386.635,A -85,B 0,C 180,E1 -9292.961,E2 -9292.961} C_VEL
LIN {X 0,Y 432.32,Z 386.632,A -85,B 0,C 180,E1 -9294.999,E2 -9294.999} C_VEL
LIN {X 0,Y 432.224,Z 386.645,A -85,B 0,C 180,E1 -9297.078,E2 -9297.078} C_VEL
LIN {X 0,Y 432.01,Z 386.673,A -85,B 0,C 180,E1 -9299.207,E2 -9299.207} C_VEL
LIN {X 0,Y 431.697,Z 386.718,A -85,B 0,C 180,E1 -9301.391,E2 -9301.391} C_VEL
LIN {X 0,Y 431.615,Z 387.441,A -85,B 0,C 180,E1 -9302.497,E2 -9302.497} C_VEL
LIN {X 0,Y 431.541,Z 390.883,A -85,B 0,C 180,E1 -9305.889,E2 -9305.889} C_VEL
LIN {X 0,Y 431.51,Z 393.668,A -85,B 0,C 180,E1 -9308.578,E2 -9308.578} C_VEL
LIN {X 0,Y 431.436,Z 396.683,A -85,B 0,C 180,E1 -9311.469,E2 -9311.469} C_VEL
LIN {X 0,Y 431.389,Z 399.865,A -85,B 0,C 180,E1 -9314.464,E2 -9314.464} C_VEL
LIN {X 0,Y 431.424,Z 401.032,A -85,B 0,C 180,E1 -9315.536,E2 -9315.536} C_VEL
LIN {X 0,Y 434.674,Z 414.942,A -85,B 0,C 180,E1 -9316.131,E2 -9316.131} C_VEL
LIN {X 0,Y 435.782,Z 420.827,A -85,B 0,C 180,E1 -9316.439,E2 -9316.439} C_VEL
LIN {X 0,Y 435.248,Z 433.597,A -85,B 0,C 180,E1 -9317.158,E2 -9317.158} C_VEL
LIN {X 0,Y 434.628,Z 445.628,A -85,B 0,C 180,E1 -9318.051,E2 -9318.051} C_VEL
LIN {X 0,Y 433.995,Z 456.004,A -85,B 0,C 180,E1 -9319.018,E2 -9319.018} C_VEL
LIN {X 0,Y 433.418,Z 465.974,A -85,B 0,C 180,E1 -9320.172,E2 -9320.172} C_VEL
LIN {X 0,Y 432.903,Z 474.533,A -85,B 0,C 180,E1 -9321.387,E2 -9321.387} C_VEL
LIN {X 0,Y 432.392,Z 482.557,A -85,B 0,C 180,E1 -9322.783,E2 -9322.783} C_VEL
LIN {X 0,Y 432.013,Z 488.901,A -85,B 0,C 180,E1 -9324.152,E2 -9324.152} C_VEL
LIN {X 0,Y 431.673,Z 494.656,A -85,B 0,C 180,E1 -9325.74,E2 -9325.74} C_VEL
LIN {X 0,Y 431.497,Z 499.341,A -85,B 0,C 180,E1 -9327.489,E2 -9327.489} C_VEL
LIN {X 0,Y 431.317,Z 501.453,A -85,B 0,C 180,E1 -9328.574,E2 -9328.574} C_VEL
LIN {X 0,Y 431.229,Z 503.082,A -85,B 0,C 180,E1 -9329.733,E2 -9329.733} C_VEL
LIN {X 0,Y 431.185,Z 503.967,A -85,B 0,C 180,E1 -9330.728,E2 -9330.728} C_VEL
LIN {X 0,Y 431.172,Z 504.402,A -85,B 0,C 180,E1 -9331.792,E2 -9331.792} C_VEL
LIN {X 0,Y 431.192,Z 504.355,A -85,B 0,C 180,E1 -9332.848,E2 -9332.848} C_VEL
LIN {X 0,Y 431.227,Z 503.757,A -85,B 0,C 180,E1 -9333.895,E2 -9333.895} C_VEL
LIN {X 0,Y 431.311,Z 502.698,A -85,B 0,C 180,E1 -9334.935,E2 -9334.935} C_VEL
LIN {X 0,Y 431.511,Z 500.163,A -85,B 0,C 180,E1 -9336.484,E2 -9336.484} C_VEL
LIN {X 0,Y 431.726,Z 496.225,A -85,B 0,C 180,E1 -9338.095,E2 -9338.095} C_VEL
LIN {X 0,Y 431.974,Z 491.53,A -85,B 0,C 180,E1 -9339.526,E2 -9339.526} C_VEL
LIN {X 0,Y 432.369,Z 485.208,A -85,B 0,C 180,E1 -9341.03,E2 -9341.03} C_VEL
LIN {X 0,Y 432.947,Z 477.266,A -85,B 0,C 180,E1 -9342.525,E2 -9342.525} C_VEL
LIN {X 0,Y 433.521,Z 468.9,A -85,B 0,C 180,E1 -9343.784,E2 -9343.784} C_VEL
LIN {X 0,Y 434.174,Z 459.048,A -85,B 0,C 180,E1 -9344.991,E2 -9344.991} C_VEL
LIN {X 0,Y 434.865,Z 448.417,A -85,B 0,C 180,E1 -9346.041,E2 -9346.041} C_VEL
LIN {X 0,Y 435.489,Z 436.864,A -85,B 0,C 180,E1 -9346.943,E2 -9346.943} C_VEL
LIN {X 0,Y 436.073,Z 424.853,A -85,B 0,C 180,E1 -9347.671,E2 -9347.671} C_VEL
LIN {X 0,Y 436.075,Z 420.239,A -85,B 0,C 180,E1 -9347.907,E2 -9347.907} C_VEL
LIN {X 0,Y 433.022,Z 407.659,A -85,B 0,C 180,E1 -9348.563,E2 -9348.563} C_VEL
LIN {X 0,Y 431.688,Z 402.767,A -85,B 0,C 180,E1 -9348.794,E2 -9348.794} C_VEL
LIN {X 0,Y 431.79,Z 399.208,A -85,B 0,C 180,E1 -9352.519,E2 -9352.519} C_VEL
LIN {X 0,Y 432.017,Z 396.549,A -85,B 0,C 180,E1 -9355.335,E2 -9355.335} C_VEL
LIN {X 0,Y 432.098,Z 393.165,A -85,B 0,C 180,E1 -9359.069,E2 -9359.069} C_VEL
LIN {X 0,Y 432.376,Z 391.496,A -85,B 0,C 180,E1 -9360.932,E2 -9360.932} C_VEL
LIN {X 0,Y 432.45,Z 387.5,A -85,B 0,C 180,E1 -9365.597,E2 -9365.597} C_VEL
LIN {X 0,Y 432.407,Z 386.742,A -85,B 0,C 180,E1 -9366.534,E2 -9366.534} C_VEL
LIN {X 0,Y 432.44,Z 386.623,A -85,B 0,C 180,E1 -9368.411,E2 -9368.411} C_VEL
LIN {X 0,Y 432.393,Z 386.626,A -85,B 0,C 180,E1 -9371.248,E2 -9371.248} C_VEL
LIN {X 0,Y 432.353,Z 386.63,A -85,B 0,C 180,E1 -9374.113,E2 -9374.113} C_VEL
LIN {X 0,Y 432.398,Z 386.624,A -85,B 0,C 180,E1 -9377.012,E2 -9377.012} C_VEL
LIN {X 0,Y 432.349,Z 386.631,A -85,B 0,C 180,E1 -9379.961,E2 -9379.961} C_VEL
LIN {X 0,Y 432.302,Z 386.634,A -85,B 0,C 180,E1 -9382.966,E2 -9382.966} C_VEL
LIN {X 0,Y 432.34,Z 386.631,A -85,B 0,C 180,E1 -9386.035,E2 -9386.035} C_VEL
LIN {X 0,Y 432.322,Z 386.634,A -85,B 0,C 180,E1 -9389.19,E2 -9389.19} C_VEL
LIN {X 0,Y 432.297,Z 386.637,A -85,B 0,C 180,E1 -9392.296,E2 -9392.296} C_VEL
LIN {X 0,Y 432.314,Z 386.635,A -85,B 0,C 180,E1 -9394.68,E2 -9394.68} C_VEL
LIN {X 0,Y 432.329,Z 386.635,A -85,B 0,C 180,E1 -9398.152,E2 -9398.152} C_VEL
LIN {X 0,Y 432.35,Z 386.634,A -85,B 0,C 180,E1 -9401.612,E2 -9401.612} C_VEL
LIN {X 0,Y 432.356,Z 386.632,A -85,B 0,C 180,E1 -9404.345,E2 -9404.345} C_VEL
LIN {X 0,Y 432.354,Z 386.722,A -85,B 0,C 180,E1 -9406.309,E2 -9406.309} C_VEL
LIN {X 0,Y 433.24,Z 391.671,A -85,B 0,C 180,E1 -9409.68,E2 -9409.68} C_VEL
LIN {X 0,Y 434.08,Z 396.46,A -85,B 0,C 180,E1 -9412.499,E2 -9412.499} C_VEL
LIN {X 0,Y 434.313,Z 399.964,A -85,B 0,C 180,E1 -9414.376,E2 -9414.376} C_VEL
LIN {X 0,Y 433.694,Z 406.311,A -85,B 0,C 180,E1 -9417.423,E2 -9417.423} C_VEL
LIN {X 0,Y 433.061,Z 412.813,A -85,B 0,C 180,E1 -9420.337,E2 -9420.337} C_VEL
LIN {X 0,Y 432.647,Z 419.815,A -85,B 0,C 180,E1 -9423.309,E2 -9423.309} C_VEL
LIN {X 0,Y 432.26,Z 427.727,A -85,B 0,C 180,E1 -9426.53,E2 -9426.53} C_VEL
LIN {X 0,Y 431.912,Z 436.675,A -85,B 0,C 180,E1 -9430.023,E2 -9430.023} C_VEL
LIN {X 0,Y 431.659,Z 445.098,A -85,B 0,C 180,E1 -9433.193,E2 -9433.193} C_VEL
LIN {X 0,Y 433.81,Z 458.71,A -85,B 0,C 180,E1 -9433.701,E2 -9433.701} C_VEL
LIN {X 0,Y 435.13,Z 472.099,A -85,B 0,C 180,E1 -9434.368,E2 -9434.368} C_VEL
LIN {X 0,Y 435.019,Z 479.285,A -85,B 0,C 180,E1 -9434.784,E2 -9434.784} C_VEL
LIN {X 0,Y 434.282,Z 490.987,A -85,B 0,C 180,E1 -9435.597,E2 -9435.597} C_VEL
LIN {X 0,Y 433.537,Z 502.028,A -85,B 0,C 180,E1 -9436.571,E2 -9436.571} C_VEL
LIN {X 0,Y 433.047,Z 511.384,A -85,B 0,C 180,E1 -9437.586,E2 -9437.586} C_VEL
LIN {X 0,Y 432.513,Z 520.341,A -85,B 0,C 180,E1 -9438.76,E2 -9438.76} C_VEL
LIN {X 0,Y 432.011,Z 527.764,A -85,B 0,C 180,E1 -9439.932,E2 -9439.932} C_VEL
LIN {X 0,Y 431.675,Z 535.105,A -85,B 0,C 180,E1 -9441.342,E2 -9441.342} C_VEL
LIN {X 0,Y 431.463,Z 540.074,A -85,B 0,C 180,E1 -9442.516,E2 -9442.516} C_VEL
LIN {X 0,Y 431.293,Z 545.198,A -85,B 0,C 180,E1 -9444.011,E2 -9444.011} C_VEL
LIN {X 0,Y 431.286,Z 548.642,A -85,B 0,C 180,E1 -9445.33,E2 -9445.33} C_VEL
LIN {X 0,Y 431.231,Z 550.555,A -85,B 0,C 180,E1 -9446.266,E2 -9446.266} C_VEL
LIN {X 0,Y 431.318,Z 552.002,A -85,B 0,C 180,E1 -9447.202,E2 -9447.202} C_VEL
LIN {X 0,Y 431.285,Z 553.037,A -85,B 0,C 180,E1 -9448.136,E2 -9448.136} C_VEL
LIN {X 0,Y 431.277,Z 553.676,A -85,B 0,C 180,E1 -9449.07,E2 -9449.07} C_VEL
LIN {X 0,Y 431.278,Z 553.896,A -85,B 0,C 180,E1 -9450.003,E2 -9450.003} C_VEL
LIN {X 0,Y 431.277,Z 553.678,A -85,B 0,C 180,E1 -9450.937,E2 -9450.937} C_VEL
LIN {X 0,Y 431.286,Z 553.066,A -85,B 0,C 180,E1 -9451.871,E2 -9451.871} C_VEL
LIN {X 0,Y 431.319,Z 552.056,A -85,B 0,C 180,E1 -9452.805,E2 -9452.805} C_VEL
LIN {X 0,Y 431.235,Z 550.602,A -85,B 0,C 180,E1 -9453.741,E2 -9453.741} C_VEL
LIN {X 0,Y 431.333,Z 547.6,A -85,B 0,C 180,E1 -9455.145,E2 -9455.145} C_VEL
LIN {X 0,Y 431.381,Z 543.516,A -85,B 0,C 180,E1 -9456.552,E2 -9456.552} C_VEL
LIN {X 0,Y 431.602,Z 537.231,A -85,B 0,C 180,E1 -9458.195,E2 -9458.195} C_VEL
LIN {X 0,Y 431.906,Z 530.383,A -85,B 0,C 180,E1 -9459.604,E2 -9459.604} C_VEL
LIN {X 0,Y 432.373,Z 521.859,A -85,B 0,C 180,E1 -9461.014,E2 -9461.014} C_VEL
LIN {X 0,Y 432.941,Z 513.102,A -85,B 0,C 180,E1 -9462.186,E2 -9462.186} C_VEL
LIN {X 0,Y 433.417,Z 503.202,A -85,B 0,C 180,E1 -9463.276,E2 -9463.276} C_VEL
LIN {X 0,Y 434.148,Z 491.678,A -85,B 0,C 180,E1 -9464.295,E2 -9464.295} C_VEL
LIN {X 0,Y 434.864,Z 479.815,A -85,B 0,C 180,E1 -9465.109,E2 -9465.109} C_VEL
LIN {X 0,Y 435.093,Z 472.502,A -85,B 0,C 180,E1 -9465.52,E2 -9465.52} C_VEL
LIN {X 0,Y 433.539,Z 459.248,A -85,B 0,C 180,E1 -9466.158,E2 -9466.158} C_VEL
LIN {X 0,Y 431.715,Z 446.61,A -85,B 0,C 180,E1 -9466.608,E2 -9466.608} C_VEL
LIN {X 0,Y 431.964,Z 437.772,A -85,B 0,C 180,E1 -9469.981,E2 -9469.981} C_VEL
LIN {X 0,Y 432.358,Z 428.811,A -85,B 0,C 180,E1 -9473.472,E2 -9473.472} C_VEL
LIN {X 0,Y 432.766,Z 420.668,A -85,B 0,C 180,E1 -9476.723,E2 -9476.723} C_VEL
LIN {X 0,Y 433.296,Z 412.206,A -85,B 0,C 180,E1 -9480.189,E2 -9480.189} C_VEL
LIN {X 0,Y 433.867,Z 404.584,A -85,B 0,C 180,E1 -9483.421,E2 -9483.421} C_VEL
LIN {X 0,Y 434.281,Z 399.501,A -85,B 0,C 180,E1 -9485.636,E2 -9485.636} C_VEL
LIN {X 0,Y 433.904,Z 395.562,A -85,B 0,C 180,E1 -9487.47,E2 -9487.47} C_VEL
LIN {X 0,Y 432.861,Z 389.328,A -85,B 0,C 180,E1 -9490.503,E2 -9490.503} C_VEL
LIN {X 0,Y 432.351,Z 386.632,A -85,B 0,C 180,E1 -9491.954,E2 -9491.954} C_VEL
LIN {X 0,Y 432.346,Z 386.631,A -85,B 0,C 180,E1 -9494.349,E2 -9494.349} C_VEL
LIN {X 0,Y 432.32,Z 386.635,A -85,B 0,C 180,E1 -9497.019,E2 -9497.019} C_VEL
LIN {X 0,Y 432.304,Z 386.636,A -85,B 0,C 180,E1 -9499.829,E2 -9499.829} C_VEL
LIN {X 0,Y 432.317,Z 386.636,A -85,B 0,C 180,E1 -9503.022,E2 -9503.022} C_VEL
LIN {X 0,Y 432.346,Z 386.629,A -85,B 0,C 180,E1 -9506.003,E2 -9506.003} C_VEL
LIN {X 0,Y 432.36,Z 386.629,A -85,B 0,C 180,E1 -9509.491,E2 -9509.491} C_VEL
LIN {X 0,Y 432.356,Z 386.629,A -85,B 0,C 180,E1 -9511.874,E2 -9511.874} C_VEL
LIN {X 0,Y 432.39,Z 386.626,A -85,B 0,C 180,E1 -9515.539,E2 -9515.539} C_VEL
LIN {X 0,Y 432.363,Z 386.63,A -85,B 0,C 180,E1 -9519.046,E2 -9519.046} C_VEL
LIN {X 0,Y 432.373,Z 386.625,A -85,B 0,C 180,E1 -9522.01,E2 -9522.01} C_VEL
LIN {X 0,Y 432.404,Z 386.624,A -85,B 0,C 180,E1 -9524.926,E2 -9524.926} C_VEL
LIN {X 0,Y 432.471,Z 386.615,A -85,B 0,C 180,E1 -9527.803,E2 -9527.803} C_VEL
LIN {X 0,Y 432.476,Z 386.615,A -85,B 0,C 180,E1 -9531.589,E2 -9531.589} C_VEL
LIN {X 0,Y 432.598,Z 386.599,A -85,B 0,C 180,E1 -9534.405,E2 -9534.405} C_VEL
LIN {X 0,Y 432.613,Z 386.596,A -85,B 0,C 180,E1 -9538.137,E2 -9538.137} C_VEL
LIN {X 0,Y 432.738,Z 386.581,A -85,B 0,C 180,E1 -9539.999,E2 -9539.999} C_VEL
LIN {X 0,Y 432.591,Z 386.603,A -85,B 0,C 180,E1 -9542.793,E2 -9542.793} C_VEL
LIN {X 0,Y 432.587,Z 386.6,A -85,B 0,C 180,E1 -9545.593,E2 -9545.593} C_VEL
LIN {X 0,Y 432.473,Z 386.616,A -85,B 0,C 180,E1 -9548.409,E2 -9548.409} C_VEL
LIN {X 0,Y 432.468,Z 386.615,A -85,B 0,C 180,E1 -9552.195,E2 -9552.195} C_VEL
LIN {X 0,Y 432.439,Z 386.618,A -85,B 0,C 180,E1 -9556.038,E2 -9556.038} C_VEL
LIN {X 0,Y 432.396,Z 386.623,A -85,B 0,C 180,E1 -9559.483,E2 -9559.483} C_VEL
LIN {X 0,Y 432.326,Z 386.635,A -85,B 0,C 180,E1 -9562.963,E2 -9562.963} C_VEL
LIN {X 0,Y 432.35,Z 386.631,A -85,B 0,C 180,E1 -9565,E2 -9565} C_VEL
LIN {X 0,Y 432.378,Z 386.626,A -85,B 0,C 180,E1 -9568.122,E2 -9568.122} C_VEL
LIN {X 0,Y 432.327,Z 386.631,A -85,B 0,C 180,E1 -9571.344,E2 -9571.344} C_VEL
LIN {X 0,Y 432.346,Z 386.632,A -85,B 0,C 180,E1 -9574.675,E2 -9574.675} C_VEL
LIN {X 0,Y 432.337,Z 386.633,A -85,B 0,C 180,E1 -9578.149,E2 -9578.149} C_VEL
LIN {X 0,Y 432.33,Z 386.632,A -85,B 0,C 180,E1 -9581.598,E2 -9581.598} C_VEL
LIN {X 0,Y 432.339,Z 386.633,A -85,B 0,C 180,E1 -9584.345,E2 -9584.345} C_VEL
LIN {X 0,Y 432.321,Z 386.634,A -85,B 0,C 180,E1 -9587.014,E2 -9587.014} C_VEL
LIN {X 0,Y 432.336,Z 386.632,A -85,B 0,C 180,E1 -9589.819,E2 -9589.819} C_VEL
LIN {X 0,Y 432.31,Z 386.635,A -85,B 0,C 180,E1 -9593.02,E2 -9593.02} C_VEL
LIN {X 0,Y 432.363,Z 386.628,A -85,B 0,C 180,E1 -9595.994,E2 -9595.994} C_VEL
LIN {X 0,Y 432.349,Z 386.629,A -85,B 0,C 180,E1 -9599.487,E2 -9599.487} C_VEL
LIN {X 0,Y 432.393,Z 386.626,A -85,B 0,C 180,E1 -9602.925,E2 -9602.925} C_VEL
LIN {X 0,Y 432.372,Z 386.629,A -85,B 0,C 180,E1 -9606.021,E2 -9606.021} C_VEL
LIN {X 0,Y 432.35,Z 386.629,A -85,B 0,C 180,E1 -9609.043,E2 -9609.043} C_VEL
LIN {X 0,Y 432.376,Z 386.627,A -85,B 0,C 180,E1 -9612.008,E2 -9612.008} C_VEL
LIN {X 0,Y 432.393,Z 386.625,A -85,B 0,C 180,E1 -9614.923,E2 -9614.923} C_VEL
LIN {X 0,Y 432.457,Z 386.617,A -85,B 0,C 180,E1 -9617.8,E2 -9617.8} C_VEL
LIN {X 0,Y 432.488,Z 386.611,A -85,B 0,C 180,E1 -9621.587,E2 -9621.587} C_VEL
LIN {X 0,Y 432.589,Z 386.603,A -85,B 0,C 180,E1 -9624.403,E2 -9624.403} C_VEL
LIN {X 0,Y 432.599,Z 386.6,A -85,B 0,C 180,E1 -9628.135,E2 -9628.135} C_VEL
LIN {X 0,Y 432.724,Z 386.586,A -85,B 0,C 180,E1 -9629.997,E2 -9629.997} C_VEL
LIN {X 0,Y 432.596,Z 386.599,A -85,B 0,C 180,E1 -9632.79,E2 -9632.79} C_VEL
LIN {X 0,Y 432.452,Z 386.616,A -85,B 0,C 180,E1 -9635.008,E2 -9635.008} C_VEL
LIN {X 0,Y 431.892,Z 386.689,A -85,B 0,C 180,E1 -9635.787,E2 -9635.787} C_VEL
LIN {X 0,Y 429.048,Z 387.04,A -85,B 0,C 180,E1 -9637.052,E2 -9637.052} C_VEL
LIN {X 0,Y 426.565,Z 387.354,A -85,B 0,C 180,E1 -9638.073,E2 -9638.073} C_VEL
LIN {X 0,Y 425.485,Z 387.485,A -85,B 0,C 180,E1 -9638.863,E2 -9638.863} C_VEL
LIN {X 0,Y 425.393,Z 387.495,A -85,B 0,C 180,E1 -9639.131,E2 -9639.131} C_VEL
LIN {X 0,Y 425.39,Z 387.496,A -85,B 0,C 180,E1 -9642.907,E2 -9642.907} C_VEL
LIN {X 0,Y 425.354,Z 387.501,A -85,B 0,C 180,E1 -9646.605,E2 -9646.605} C_VEL
LIN {X 0,Y 425.311,Z 387.507,A -85,B 0,C 180,E1 -9649.632,E2 -9649.632} C_VEL
LIN {X 0,Y 425.289,Z 387.51,A -85,B 0,C 180,E1 -9653.362,E2 -9653.362} C_VEL
LIN {X 0,Y 425.252,Z 387.515,A -85,B 0,C 180,E1 -9656.497,E2 -9656.497} C_VEL
LIN {X 0,Y 425.014,Z 387.544,A -85,B 0,C 180,E1 -9658.791,E2 -9658.791} C_VEL
LIN {X 0,Y 424.596,Z 387.643,A -85,B 0,C 180,E1 -9661.978,E2 -9661.978} C_VEL
LIN {X 0,Y 424.502,Z 391.077,A -85,B 0,C 180,E1 -9665.407,E2 -9665.407} C_VEL
LIN {X 0,Y 424.456,Z 393.504,A -85,B 0,C 180,E1 -9667.774,E2 -9667.774} C_VEL
LIN {X 0,Y 424.416,Z 396.211,A -85,B 0,C 180,E1 -9670.385,E2 -9670.385} C_VEL
LIN {X 0,Y 424.335,Z 400.094,A -85,B 0,C 180,E1 -9674.07,E2 -9674.07} C_VEL
LIN {X 0,Y 424.365,Z 401.603,A -85,B 0,C 180,E1 -9675.29,E2 -9675.29} C_VEL
LIN {X 0,Y 427.64,Z 415.43,A -85,B 0,C 180,E1 -9675.898,E2 -9675.898} C_VEL
LIN {X 0,Y 428.876,Z 421.598,A -85,B 0,C 180,E1 -9676.231,E2 -9676.231} C_VEL
LIN {X 0,Y 428.422,Z 433.248,A -85,B 0,C 180,E1 -9676.896,E2 -9676.896} C_VEL
LIN {X 0,Y 427.74,Z 445.518,A -85,B 0,C 180,E1 -9677.811,E2 -9677.811} C_VEL
LIN {X 0,Y 427.059,Z 456.381,A -85,B 0,C 180,E1 -9678.833,E2 -9678.833} C_VEL
LIN {X 0,Y 426.449,Z 466.355,A -85,B 0,C 180,E1 -9680.006,E2 -9680.006} C_VEL
LIN {X 0,Y 425.924,Z 474.486,A -85,B 0,C 180,E1 -9681.171,E2 -9681.171} C_VEL
LIN {X 0,Y 425.43,Z 481.885,A -85,B 0,C 180,E1 -9682.454,E2 -9682.454} C_VEL
LIN {X 0,Y 425.025,Z 488.404,A -85,B 0,C 180,E1 -9683.84,E2 -9683.84} C_VEL
LIN {X 0,Y 424.745,Z 493.519,A -85,B 0,C 180,E1 -9685.192,E2 -9685.192} C_VEL
LIN {X 0,Y 424.475,Z 498.47,A -85,B 0,C 180,E1 -9686.882,E2 -9686.882} C_VEL
LIN {X 0,Y 424.339,Z 500.876,A -85,B 0,C 180,E1 -9687.996,E2 -9687.996} C_VEL
LIN {X 0,Y 424.154,Z 503.204,A -85,B 0,C 180,E1 -9689.488,E2 -9689.488} C_VEL
LIN {X 0,Y 424.107,Z 504.731,A -85,B 0,C 180,E1 -9691.425,E2 -9691.425} C_VEL
LIN {X 0,Y 424.081,Z 504.847,A -85,B 0,C 180,E1 -9692.354,E2 -9692.354} C_VEL
LIN {X 0,Y 424.116,Z 504.502,A -85,B 0,C 180,E1 -9693.475,E2 -9693.475} C_VEL
LIN {X 0,Y 424.198,Z 503.711,A -85,B 0,C 180,E1 -9694.485,E2 -9694.485} C_VEL
LIN {X 0,Y 424.302,Z 502.236,A -85,B 0,C 180,E1 -9695.632,E2 -9695.632} C_VEL
LIN {X 0,Y 424.539,Z 499.446,A -85,B 0,C 180,E1 -9697.107,E2 -9697.107} C_VEL
LIN {X 0,Y 424.753,Z 495.367,A -85,B 0,C 180,E1 -9698.654,E2 -9698.654} C_VEL
LIN {X 0,Y 425.107,Z 490.339,A -85,B 0,C 180,E1 -9700.102,E2 -9700.102} C_VEL
LIN {X 0,Y 425.584,Z 483.128,A -85,B 0,C 180,E1 -9701.715,E2 -9701.715} C_VEL
LIN {X 0,Y 426.202,Z 474.977,A -85,B 0,C 180,E1 -9703.159,E2 -9703.159} C_VEL
LIN {X 0,Y 426.908,Z 465.657,A -85,B 0,C 180,E1 -9704.484,E2 -9704.484} C_VEL
LIN {X 0,Y 427.616,Z 454.757,A -85,B 0,C 180,E1 -9705.729,E2 -9705.729} C_VEL
LIN {X 0,Y 428.372,Z 443.812,A -85,B 0,C 180,E1 -9706.722,E2 -9706.722} C_VEL
LIN {X 0,Y 428.951,Z 432.675,A -85,B 0,C 180,E1 -9707.523,E2 -9707.523} C_VEL
LIN {X 0,Y 429.446,Z 422.907,A -85,B 0,C 180,E1 -9708.077,E2 -9708.077} C_VEL
LIN {X 0,Y 427,Z 411.626,A -85,B 0,C 180,E1 -9708.7,E2 -9708.7} C_VEL
LIN {X 0,Y 424.628,Z 403.241,A -85,B 0,C 180,E1 -9709.119,E2 -9709.119} C_VEL
LIN {X 0,Y 424.777,Z 399.556,A -85,B 0,C 180,E1 -9713.033,E2 -9713.033} C_VEL
LIN {X 0,Y 424.981,Z 397.502,A -85,B 0,C 180,E1 -9715.258,E2 -9715.258} C_VEL
LIN {X 0,Y 425.142,Z 393.29,A -85,B 0,C 180,E1 -9720.001,E2 -9720.001} C_VEL
LIN {X 0,Y 425.343,Z 392.43,A -85,B 0,C 180,E1 -9720.948,E2 -9720.948} C_VEL
LIN {X 0,Y 425.43,Z 388.469,A -85,B 0,C 180,E1 -9725.689,E2 -9725.689} C_VEL
LIN {X 0,Y 425.401,Z 387.71,A -85,B 0,C 180,E1 -9726.642,E2 -9726.642} C_VEL
LIN {X 0,Y 425.397,Z 387.501,A -85,B 0,C 180,E1 -9728.552,E2 -9728.552} C_VEL
LIN {X 0,Y 425.351,Z 387.504,A -85,B 0,C 180,E1 -9731.437,E2 -9731.437} C_VEL
LIN {X 0,Y 425.324,Z 387.506,A -85,B 0,C 180,E1 -9734.352,E2 -9734.352} C_VEL
LIN {X 0,Y 425.332,Z 387.505,A -85,B 0,C 180,E1 -9737.304,E2 -9737.304} C_VEL
LIN {X 0,Y 425.294,Z 387.51,A -85,B 0,C 180,E1 -9740.306,E2 -9740.306} C_VEL
LIN {X 0,Y 425.286,Z 387.51,A -85,B 0,C 180,E1 -9743.367,E2 -9743.367} C_VEL
LIN {X 0,Y 425.321,Z 387.508,A -85,B 0,C 180,E1 -9746.848,E2 -9746.848} C_VEL
LIN {X 0,Y 425.289,Z 387.51,A -85,B 0,C 180,E1 -9749.72,E2 -9749.72} C_VEL
LIN {X 0,Y 425.254,Z 387.515,A -85,B 0,C 180,E1 -9753.051,E2 -9753.051} C_VEL
LIN {X 0,Y 425.259,Z 387.514,A -85,B 0,C 180,E1 -9755.933,E2 -9755.933} C_VEL
LIN {X 0,Y 425.291,Z 387.512,A -85,B 0,C 180,E1 -9759.05,E2 -9759.05} C_VEL
LIN {X 0,Y 425.309,Z 387.51,A -85,B 0,C 180,E1 -9762.65,E2 -9762.65} C_VEL
LIN {X 0,Y 425.335,Z 387.579,A -85,B 0,C 180,E1 -9765.757,E2 -9765.757} C_VEL
LIN {X 0,Y 426.205,Z 392.655,A -85,B 0,C 180,E1 -9769.335,E2 -9769.335} C_VEL
LIN {X 0,Y 427.122,Z 397.822,A -85,B 0,C 180,E1 -9772.502,E2 -9772.502} C_VEL
LIN {X 0,Y 427.352,Z 401.097,A -85,B 0,C 180,E1 -9774.286,E2 -9774.286} C_VEL
LIN {X 0,Y 426.752,Z 406.863,A -85,B 0,C 180,E1 -9777.13,E2 -9777.13} C_VEL
LIN {X 0,Y 426.048,Z 413.868,A -85,B 0,C 180,E1 -9780.344,E2 -9780.344} C_VEL
LIN {X 0,Y 425.595,Z 421.216,A -85,B 0,C 180,E1 -9783.526,E2 -9783.526} C_VEL
LIN {X 0,Y 425.135,Z 429.979,A -85,B 0,C 180,E1 -9787.144,E2 -9787.144} C_VEL
LIN {X 0,Y 424.776,Z 438.91,A -85,B 0,C 180,E1 -9790.681,E2 -9790.681} C_VEL
LIN {X 0,Y 424.611,Z 444.559,A -85,B 0,C 180,E1 -9792.857,E2 -9792.857} C_VEL
LIN {X 0,Y 426.967,Z 459.295,A -85,B 0,C 180,E1 -9793.442,E2 -9793.442} C_VEL
LIN {X 0,Y 428.287,Z 473.169,A -85,B 0,C 180,E1 -9794.173,E2 -9794.173} C_VEL
LIN {X 0,Y 427.807,Z 484.472,A -85,B 0,C 180,E1 -9794.887,E2 -9794.887} C_VEL
LIN {X 0,Y 427.025,Z 496.305,A -85,B 0,C 180,E1 -9795.833,E2 -9795.833} C_VEL
LIN {X 0,Y 426.251,Z 506.974,A -85,B 0,C 180,E1 -9796.901,E2 -9796.901} C_VEL
LIN {X 0,Y 425.737,Z 516.667,A -85,B 0,C 180,E1 -9798.096,E2 -9798.096} C_VEL
LIN {X 0,Y 425.033,Z 526.04,A -85,B 0,C 180,E1 -9799.524,E2 -9799.524} C_VEL
LIN {X 0,Y 424.644,Z 533.612,A -85,B 0,C 180,E1 -9800.958,E2 -9800.958} C_VEL
LIN {X 0,Y 424.383,Z 539.714,A -85,B 0,C 180,E1 -9802.391,E2 -9802.391} C_VEL
LIN {X 0,Y 424.246,Z 544.169,A -85,B 0,C 180,E1 -9803.7,E2 -9803.7} C_VEL
LIN {X 0,Y 424.217,Z 548.255,A -85,B 0,C 180,E1 -9805.252,E2 -9805.252} C_VEL
LIN {X 0,Y 424.139,Z 550.159,A -85,B 0,C 180,E1 -9806.203,E2 -9806.203} C_VEL
LIN {X 0,Y 424.227,Z 551.603,A -85,B 0,C 180,E1 -9807.155,E2 -9807.155} C_VEL
LIN {X 0,Y 424.207,Z 552.637,A -85,B 0,C 180,E1 -9808.105,E2 -9808.105} C_VEL
LIN {X 0,Y 424.19,Z 553.273,A -85,B 0,C 180,E1 -9809.054,E2 -9809.054} C_VEL
LIN {X 0,Y 424.203,Z 553.485,A -85,B 0,C 180,E1 -9810.003,E2 -9810.003} C_VEL
LIN {X 0,Y 424.191,Z 553.263,A -85,B 0,C 180,E1 -9810.953,E2 -9810.953} C_VEL
LIN {X 0,Y 424.208,Z 552.648,A -85,B 0,C 180,E1 -9811.902,E2 -9811.902} C_VEL
LIN {X 0,Y 424.247,Z 551.634,A -85,B 0,C 180,E1 -9812.852,E2 -9812.852} C_VEL
LIN {X 0,Y 424.143,Z 550.166,A -85,B 0,C 180,E1 -9813.804,E2 -9813.804} C_VEL
LIN {X 0,Y 424.244,Z 547.151,A -85,B 0,C 180,E1 -9815.231,E2 -9815.231} C_VEL
LIN {X 0,Y 424.304,Z 543.052,A -85,B 0,C 180,E1 -9816.661,E2 -9816.661} C_VEL
LIN {X 0,Y 424.527,Z 536.747,A -85,B 0,C 180,E1 -9818.332,E2 -9818.332} C_VEL
LIN {X 0,Y 424.865,Z 529.88,A -85,B 0,C 180,E1 -9819.765,E2 -9819.765} C_VEL
LIN {X 0,Y 425.247,Z 522.876,A -85,B 0,C 180,E1 -9820.959,E2 -9820.959} C_VEL
LIN {X 0,Y 425.861,Z 514.46,A -85,B 0,C 180,E1 -9822.15,E2 -9822.15} C_VEL
LIN {X 0,Y 426.374,Z 504.075,A -85,B 0,C 180,E1 -9823.345,E2 -9823.345} C_VEL
LIN {X 0,Y 427.132,Z 492.45,A -85,B 0,C 180,E1 -9824.413,E2 -9824.413} C_VEL
LIN {X 0,Y 427.867,Z 481.002,A -85,B 0,C 180,E1 -9825.24,E2 -9825.24} C_VEL
LIN {X 0,Y 428.1,Z 472.782,A -85,B 0,C 180,E1 -9825.719,E2 -9825.719} C_VEL
LIN {X 0,Y 426.579,Z 459.588,A -85,B 0,C 180,E1 -9826.376,E2 -9826.376} C_VEL
LIN {X 0,Y 424.632,Z 446.287,A -85,B 0,C 180,E1 -9826.855,E2 -9826.855} C_VEL
LIN {X 0,Y 424.906,Z 437.39,A -85,B 0,C 180,E1 -9830.328,E2 -9830.328} C_VEL
LIN {X 0,Y 425.275,Z 429.744,A -85,B 0,C 180,E1 -9833.37,E2 -9833.37} C_VEL
LIN {X 0,Y 425.658,Z 422.088,A -85,B 0,C 180,E1 -9836.477,E2 -9836.477} C_VEL
LIN {X 0,Y 426.193,Z 414.467,A -85,B 0,C 180,E1 -9839.653,E2 -9839.653} C_VEL
LIN {X 0,Y 426.758,Z 406.839,A -85,B 0,C 180,E1 -9842.922,E2 -9842.922} C_VEL
LIN {X 0,Y 427.275,Z 401.784,A -85,B 0,C 180,E1 -9845.151,E2 -9845.151} C_VEL
LIN {X 0,Y 427.112,Z 397.965,A -85,B 0,C 180,E1 -9846.916,E2 -9846.916} C_VEL
LIN {X 0,Y 426.069,Z 391.606,A -85,B 0,C 180,E1 -9850.042,E2 -9850.042} C_VEL
LIN {X 0,Y 425.322,Z 387.507,A -85,B 0,C 180,E1 -9852.263,E2 -9852.263} C_VEL
LIN {X 0,Y 425.297,Z 387.507,A -85,B 0,C 180,E1 -9855.284,E2 -9855.284} C_VEL
LIN {X 0,Y 425.265,Z 387.514,A -85,B 0,C 180,E1 -9858.619,E2 -9858.619} C_VEL
LIN {X 0,Y 425.294,Z 387.511,A -85,B 0,C 180,E1 -9861.1,E2 -9861.1} C_VEL
LIN {X 0,Y 425.308,Z 387.507,A -85,B 0,C 180,E1 -9864.664,E2 -9864.664} C_VEL
LIN {X 0,Y 425.276,Z 387.51,A -85,B 0,C 180,E1 -9868.073,E2 -9868.073} C_VEL
LIN {X 0,Y 425.324,Z 387.506,A -85,B 0,C 180,E1 -9871.367,E2 -9871.367} C_VEL
LIN {X 0,Y 425.281,Z 387.51,A -85,B 0,C 180,E1 -9874.553,E2 -9874.553} C_VEL
LIN {X 0,Y 425.297,Z 387.509,A -85,B 0,C 180,E1 -9876.634,E2 -9876.634} C_VEL
LIN {X 0,Y 425.308,Z 387.507,A -85,B 0,C 180,E1 -9879.694,E2 -9879.694} C_VEL
LIN {X 0,Y 425.346,Z 387.503,A -85,B 0,C 180,E1 -9882.697,E2 -9882.697} C_VEL
LIN {X 0,Y 425.357,Z 387.5,A -85,B 0,C 180,E1 -9885.65,E2 -9885.65} C_VEL
LIN {X 0,Y 425.359,Z 387.502,A -85,B 0,C 180,E1 -9888.563,E2 -9888.563} C_VEL
LIN {X 0,Y 425.519,Z 387.481,A -85,B 0,C 180,E1 -9892.31,E2 -9892.31} C_VEL
LIN {X 0,Y 425.554,Z 387.476,A -85,B 0,C 180,E1 -9894.312,E2 -9894.312} C_VEL
LIN {X 0,Y 425.582,Z 387.472,A -85,B 0,C 180,E1 -9898.106,E2 -9898.106} C_VEL
LIN {X 0,Y 425.707,Z 387.456,A -85,B 0,C 180,E1 -9899.999,E2 -9899.999} C_VEL
LIN {X 0,Y 425.545,Z 387.481,A -85,B 0,C 180,E1 -9902.839,E2 -9902.839} C_VEL
LIN {X 0,Y 425.541,Z 387.477,A -85,B 0,C 180,E1 -9905.686,E2 -9905.686} C_VEL
LIN {X 0,Y 425.418,Z 387.496,A -85,B 0,C 180,E1 -9908.55,E2 -9908.55} C_VEL
LIN {X 0,Y 425.422,Z 387.494,A -85,B 0,C 180,E1 -9912.401,E2 -9912.401} C_VEL
LIN {X 0,Y 425.397,Z 387.497,A -85,B 0,C 180,E1 -9916.31,E2 -9916.31} C_VEL
LIN {X 0,Y 425.338,Z 387.502,A -85,B 0,C 180,E1 -9919.634,E2 -9919.634} C_VEL
LIN {X 0,Y 425.297,Z 387.509,A -85,B 0,C 180,E1 -9922.337,E2 -9922.337} C_VEL
LIN {X 0,Y 425.329,Z 387.506,A -85,B 0,C 180,E1 -9924.655,E2 -9924.655} C_VEL
LIN {X 0,Y 425.345,Z 387.5,A -85,B 0,C 180,E1 -9927.557,E2 -9927.557} C_VEL
LIN {X 0,Y 425.295,Z 387.512,A -85,B 0,C 180,E1 -9930.814,E2 -9930.814} C_VEL
LIN {X 0,Y 425.318,Z 387.507,A -85,B 0,C 180,E1 -9934.286,E2 -9934.286} C_VEL
LIN {X 0,Y 425.282,Z 387.51,A -85,B 0,C 180,E1 -9937.693,E2 -9937.693} C_VEL
LIN {X 0,Y 425.272,Z 387.514,A -85,B 0,C 180,E1 -9940.516,E2 -9940.516} C_VEL
LIN {X 0,Y 425.26,Z 387.512,A -85,B 0,C 180,E1 -9943.348,E2 -9943.348} C_VEL
LIN {X 0,Y 425.266,Z 387.514,A -85,B 0,C 180,E1 -9946.042,E2 -9946.042} C_VEL
LIN {X 0,Y 425.28,Z 387.51,A -85,B 0,C 180,E1 -9949.478,E2 -9949.478} C_VEL
LIN {X 0,Y 425.281,Z 387.513,A -85,B 0,C 180,E1 -9952.486,E2 -9952.486} C_VEL
LIN {X 0,Y 425.311,Z 387.507,A -85,B 0,C 180,E1 -9955.815,E2 -9955.815} C_VEL
LIN {X 0,Y 425.293,Z 387.508,A -85,B 0,C 180,E1 -9959.236,E2 -9959.236} C_VEL
LIN {X 0,Y 425.351,Z 387.503,A -85,B 0,C 180,E1 -9962.439,E2 -9962.439} C_VEL
LIN {X 0,Y 425.352,Z 387.5,A -85,B 0,C 180,E1 -9965.599,E2 -9965.599} C_VEL
LIN {X 0,Y 425.293,Z 387.51,A -85,B 0,C 180,E1 -9968.679,E2 -9968.679} C_VEL
LIN {X 0,Y 425.331,Z 387.505,A -85,B 0,C 180,E1 -9971.7,E2 -9971.7} C_VEL
LIN {X 0,Y 425.346,Z 387.503,A -85,B 0,C 180,E1 -9974.668,E2 -9974.668} C_VEL
LIN {X 0,Y 425.409,Z 387.493,A -85,B 0,C 180,E1 -9977.595,E2 -9977.595} C_VEL
LIN {X 0,Y 425.438,Z 387.489,A -85,B 0,C 180,E1 -9981.447,E2 -9981.447} C_VEL
LIN {X 0,Y 425.545,Z 387.48,A -85,B 0,C 180,E1 -9984.31,E2 -9984.31} C_VEL
LIN {X 0,Y 425.568,Z 387.476,A -85,B 0,C 180,E1 -9988.104,E2 -9988.104} C_VEL
LIN {X 0,Y 425.694,Z 387.461,A -85,B 0,C 180,E1 -9989.997,E2 -9989.997} C_VEL
LIN {X 0,Y 425.548,Z 387.476,A -85,B 0,C 180,E1 -9992.836,E2 -9992.836} C_VEL
LIN {X 0,Y 425.521,Z 387.481,A -85,B 0,C 180,E1 -9996.635,E2 -9996.635} C_VEL
LIN {X 0,Y 425.393,Z 387.495,A -85,B 0,C 180,E1 -9999.131,E2 -9999.131} C_VEL
LIN {X 0,Y 424.722,Z 387.582,A -85,B 0,C 180,E1 -9999.921,E2 -9999.921} C_VEL
LIN {X 0,Y 421.876,Z 387.934,A -85,B 0,C 180,E1 -10001.205,E2 -10001.205} C_VEL
LIN {X 0,Y 419.462,Z 388.237,A -85,B 0,C 180,E1 -10002.241,E2 -10002.241} C_VEL
LIN {X 0,Y 418.413,Z 388.365,A -85,B 0,C 180,E1 -10003.042,E2 -10003.042} C_VEL
LIN {X 0,Y 418.321,Z 388.377,A -85,B 0,C 180,E1 -10003.313,E2 -10003.313} C_VEL
LIN {X 0,Y 418.304,Z 388.379,A -85,B 0,C 180,E1 -10006.735,E2 -10006.735} C_VEL
LIN {X 0,Y 418.254,Z 388.387,A -85,B 0,C 180,E1 -10009.787,E2 -10009.787} C_VEL
LIN {X 0,Y 418.22,Z 388.39,A -85,B 0,C 180,E1 -10012.733,E2 -10012.733} C_VEL
LIN {X 0,Y 418.204,Z 388.394,A -85,B 0,C 180,E1 -10015.904,E2 -10015.904} C_VEL
LIN {X 0,Y 417.932,Z 388.426,A -85,B 0,C 180,E1 -10019.024,E2 -10019.024} C_VEL
LIN {X 0,Y 417.606,Z 388.473,A -85,B 0,C 180,E1 -10021.442,E2 -10021.442} C_VEL
LIN {X 0,Y 417.504,Z 389.071,A -85,B 0,C 180,E1 -10022.685,E2 -10022.685} C_VEL
LIN {X 0,Y 417.407,Z 392.493,A -85,B 0,C 180,E1 -10026.102,E2 -10026.102} C_VEL
LIN {X 0,Y 417.345,Z 395.679,A -85,B 0,C 180,E1 -10029.23,E2 -10029.23} C_VEL
LIN {X 0,Y 417.281,Z 398.922,A -85,B 0,C 180,E1 -10032.346,E2 -10032.346} C_VEL
LIN {X 0,Y 417.252,Z 401.753,A -85,B 0,C 180,E1 -10035.019,E2 -10035.019} C_VEL
LIN {X 0,Y 420.518,Z 415.504,A -85,B 0,C 180,E1 -10035.636,E2 -10035.636} C_VEL
LIN {X 0,Y 421.932,Z 421.958,A -85,B 0,C 180,E1 -10035.995,E2 -10035.995} C_VEL
LIN {X 0,Y 421.493,Z 434.299,A -85,B 0,C 180,E1 -10036.721,E2 -10036.721} C_VEL
LIN {X 0,Y 420.822,Z 446.196,A -85,B 0,C 180,E1 -10037.631,E2 -10037.631} C_VEL
LIN {X 0,Y 420.136,Z 456.458,A -85,B 0,C 180,E1 -10038.613,E2 -10038.613} C_VEL
LIN {X 0,Y 419.478,Z 466.718,A -85,B 0,C 180,E1 -10039.833,E2 -10039.833} C_VEL
LIN {X 0,Y 418.93,Z 474.858,A -85,B 0,C 180,E1 -10041.017,E2 -10041.017} C_VEL
LIN {X 0,Y 418.366,Z 482.911,A -85,B 0,C 180,E1 -10042.448,E2 -10042.448} C_VEL
LIN {X 0,Y 417.953,Z 489.698,A -85,B 0,C 180,E1 -10043.948,E2 -10043.948} C_VEL
LIN {X 0,Y 417.575,Z 495.343,A -85,B 0,C 180,E1 -10045.549,E2 -10045.549} C_VEL
LIN {X 0,Y 417.341,Z 500.155,A -85,B 0,C 180,E1 -10047.394,E2 -10047.394} C_VEL
LIN {X 0,Y 417.094,Z 503.322,A -85,B 0,C 180,E1 -10049.233,E2 -10049.233} C_VEL
LIN {X 0,Y 417.021,Z 505.035,A -85,B 0,C 180,E1 -10051.194,E2 -10051.194} C_VEL
LIN {X 0,Y 417.029,Z 505.035,A -85,B 0,C 180,E1 -10053.265,E2 -10053.265} C_VEL
LIN {X 0,Y 417.168,Z 503.524,A -85,B 0,C 180,E1 -10055.092,E2 -10055.092} C_VEL
LIN {X 0,Y 417.395,Z 500.982,A -85,B 0,C 180,E1 -10056.692,E2 -10056.692} C_VEL
LIN {X 0,Y 417.638,Z 497.276,A -85,B 0,C 180,E1 -10058.272,E2 -10058.272} C_VEL
LIN {X 0,Y 417.952,Z 492.319,A -85,B 0,C 180,E1 -10059.837,E2 -10059.837} C_VEL
LIN {X 0,Y 418.433,Z 485.992,A -85,B 0,C 180,E1 -10061.391,E2 -10061.391} C_VEL
LIN {X 0,Y 419.08,Z 478.24,A -85,B 0,C 180,E1 -10062.902,E2 -10062.902} C_VEL
LIN {X 0,Y 419.728,Z 469.848,A -85,B 0,C 180,E1 -10064.212,E2 -10064.212} C_VEL
LIN {X 0,Y 420.464,Z 459.847,A -85,B 0,C 180,E1 -10065.481,E2 -10065.481} C_VEL
LIN {X 0,Y 421.185,Z 450.015,A -85,B 0,C 180,E1 -10066.491,E2 -10066.491} C_VEL
LIN {X 0,Y 421.844,Z 439.461,A -85,B 0,C 180,E1 -10067.37,E2 -10067.37} C_VEL
LIN {X 0,Y 422.536,Z 426.841,A -85,B 0,C 180,E1 -10068.184,E2 -10068.184} C_VEL
LIN {X 0,Y 422.616,Z 423.492,A -85,B 0,C 180,E1 -10068.368,E2 -10068.368} C_VEL
LIN {X 0,Y 419.811,Z 411.502,A -85,B 0,C 180,E1 -10069.054,E2 -10069.054} C_VEL
LIN {X 0,Y 417.561,Z 403.738,A -85,B 0,C 180,E1 -10069.454,E2 -10069.454} C_VEL
LIN {X 0,Y 417.732,Z 400.225,A -85,B 0,C 180,E1 -10073.238,E2 -10073.238} C_VEL
LIN {X 0,Y 417.944,Z 398.458,A -85,B 0,C 180,E1 -10075.178,E2 -10075.178} C_VEL
LIN {X 0,Y 418.126,Z 394.222,A -85,B 0,C 180,E1 -10080.001,E2 -10080.001} C_VEL
LIN {X 0,Y 418.31,Z 393.406,A -85,B 0,C 180,E1 -10080.964,E2 -10080.964} C_VEL
LIN {X 0,Y 418.413,Z 389.441,A -85,B 0,C 180,E1 -10085.785,E2 -10085.785} C_VEL
LIN {X 0,Y 418.395,Z 388.692,A -85,B 0,C 180,E1 -10086.753,E2 -10086.753} C_VEL
LIN {X 0,Y 418.36,Z 388.377,A -85,B 0,C 180,E1 -10088.697,E2 -10088.697} C_VEL
LIN {X 0,Y 418.31,Z 388.382,A -85,B 0,C 180,E1 -10091.632,E2 -10091.632} C_VEL
LIN {X 0,Y 418.278,Z 388.385,A -85,B 0,C 180,E1 -10094.599,E2 -10094.599} C_VEL
LIN {X 0,Y 418.271,Z 388.386,A -85,B 0,C 180,E1 -10097.605,E2 -10097.605} C_VEL
LIN {X 0,Y 418.246,Z 388.389,A -85,B 0,C 180,E1 -10100.664,E2 -10100.664} C_VEL
LIN {X 0,Y 418.264,Z 388.386,A -85,B 0,C 180,E1 -10103.783,E2 -10103.783} C_VEL
LIN {X 0,Y 418.279,Z 388.383,A -85,B 0,C 180,E1 -10107.073,E2 -10107.073} C_VEL
LIN {X 0,Y 418.231,Z 388.389,A -85,B 0,C 180,E1 -10110.274,E2 -10110.274} C_VEL
LIN {X 0,Y 418.221,Z 388.392,A -85,B 0,C 180,E1 -10113.68,E2 -10113.68} C_VEL
LIN {X 0,Y 418.222,Z 388.391,A -85,B 0,C 180,E1 -10117.227,E2 -10117.227} C_VEL
LIN {X 0,Y 418.243,Z 388.389,A -85,B 0,C 180,E1 -10119.684,E2 -10119.684} C_VEL
LIN {X 0,Y 418.262,Z 388.387,A -85,B 0,C 180,E1 -10122.333,E2 -10122.333} C_VEL
LIN {X 0,Y 418.284,Z 388.452,A -85,B 0,C 180,E1 -10125.188,E2 -10125.188} C_VEL
LIN {X 0,Y 418.871,Z 391.972,A -85,B 0,C 180,E1 -10127.851,E2 -10127.851} C_VEL
LIN {X 0,Y 419.754,Z 396.881,A -85,B 0,C 180,E1 -10131.113,E2 -10131.113} C_VEL
LIN {X 0,Y 420.34,Z 400.732,A -85,B 0,C 180,E1 -10133.375,E2 -10133.375} C_VEL
LIN {X 0,Y 420.137,Z 404.458,A -85,B 0,C 180,E1 -10135.343,E2 -10135.343} C_VEL
LIN {X 0,Y 419.383,Z 411.413,A -85,B 0,C 180,E1 -10138.723,E2 -10138.723} C_VEL
LIN {X 0,Y 418.764,Z 418.591,A -85,B 0,C 180,E1 -10141.976,E2 -10141.976} C_VEL
LIN {X 0,Y 418.299,Z 425.954,A -85,B 0,C 180,E1 -10145.168,E2 -10145.168} C_VEL
LIN {X 0,Y 417.946,Z 433.496,A -85,B 0,C 180,E1 -10148.292,E2 -10148.292} C_VEL
LIN {X 0,Y 417.612,Z 441.158,A -85,B 0,C 180,E1 -10151.356,E2 -10151.356} C_VEL
LIN {X 0,Y 417.506,Z 444.177,A -85,B 0,C 180,E1 -10152.53,E2 -10152.53} C_VEL
LIN {X 0,Y 419.87,Z 457.971,A -85,B 0,C 180,E1 -10153.083,E2 -10153.083} C_VEL
LIN {X 0,Y 421.217,Z 471.105,A -85,B 0,C 180,E1 -10153.775,E2 -10153.775} C_VEL
LIN {X 0,Y 421.426,Z 477.277,A -85,B 0,C 180,E1 -10154.156,E2 -10154.156} C_VEL
LIN {X 0,Y 420.618,Z 489.163,A -85,B 0,C 180,E1 -10154.994,E2 -10154.994} C_VEL
LIN {X 0,Y 419.833,Z 499.951,A -85,B 0,C 180,E1 -10155.957,E2 -10155.957} C_VEL
LIN {X 0,Y 419.144,Z 509.102,A -85,B 0,C 180,E1 -10156.954,E2 -10156.954} C_VEL
LIN {X 0,Y 418.617,Z 518.044,A -85,B 0,C 180,E1 -10158.136,E2 -10158.136} C_VEL
LIN {X 0,Y 417.923,Z 527.087,A -85,B 0,C 180,E1 -10159.589,E2 -10159.589} C_VEL
LIN {X 0,Y 417.539,Z 534.398,A -85,B 0,C 180,E1 -10161.047,E2 -10161.047} C_VEL
LIN {X 0,Y 417.33,Z 539.357,A -85,B 0,C 180,E1 -10162.261,E2 -10162.261} C_VEL
LIN {X 0,Y 417.148,Z 544.235,A -85,B 0,C 180,E1 -10163.734,E2 -10163.734} C_VEL
LIN {X 0,Y 417.147,Z 547.881,A -85,B 0,C 180,E1 -10165.171,E2 -10165.171} C_VEL
LIN {X 0,Y 417.051,Z 549.772,A -85,B 0,C 180,E1 -10166.139,E2 -10166.139} C_VEL
LIN {X 0,Y 417.124,Z 551.21,A -85,B 0,C 180,E1 -10167.106,E2 -10167.106} C_VEL
LIN {X 0,Y 417.131,Z 552.241,A -85,B 0,C 180,E1 -10168.073,E2 -10168.073} C_VEL
LIN {X 0,Y 417.107,Z 552.872,A -85,B 0,C 180,E1 -10169.038,E2 -10169.038} C_VEL
LIN {X 0,Y 417.117,Z 553.069,A -85,B 0,C 180,E1 -10170.004,E2 -10170.004} C_VEL
LIN {X 0,Y 417.108,Z 552.842,A -85,B 0,C 180,E1 -10170.969,E2 -10170.969} C_VEL
LIN {X 0,Y 417.133,Z 552.22,A -85,B 0,C 180,E1 -10171.935,E2 -10171.935} C_VEL
LIN {X 0,Y 417.157,Z 551.199,A -85,B 0,C 180,E1 -10172.901,E2 -10172.901} C_VEL
LIN {X 0,Y 417.055,Z 549.713,A -85,B 0,C 180,E1 -10173.868,E2 -10173.868} C_VEL
LIN {X 0,Y 417.157,Z 546.678,A -85,B 0,C 180,E1 -10175.32,E2 -10175.32} C_VEL
LIN {X 0,Y 417.236,Z 542.556,A -85,B 0,C 180,E1 -10176.775,E2 -10176.775} C_VEL
LIN {X 0,Y 417.469,Z 536.224,A -85,B 0,C 180,E1 -10178.474,E2 -10178.474} C_VEL
LIN {X 0,Y 417.82,Z 529.323,A -85,B 0,C 180,E1 -10179.931,E2 -10179.931} C_VEL
LIN {X 0,Y 418.246,Z 522.282,A -85,B 0,C 180,E1 -10181.145,E2 -10181.145} C_VEL
LIN {X 0,Y 418.849,Z 513.815,A -85,B 0,C 180,E1 -10182.356,E2 -10182.356} C_VEL
LIN {X 0,Y 419.461,Z 502.675,A -85,B 0,C 180,E1 -10183.642,E2 -10183.642} C_VEL
LIN {X 0,Y 420.205,Z 491.68,A -85,B 0,C 180,E1 -10184.656,E2 -10184.656} C_VEL
LIN {X 0,Y 420.995,Z 480.101,A -85,B 0,C 180,E1 -10185.495,E2 -10185.495} C_VEL
LIN {X 0,Y 421.102,Z 473.146,A -85,B 0,C 180,E1 -10185.912,E2 -10185.912} C_VEL
LIN {X 0,Y 419.563,Z 459.654,A -85,B 0,C 180,E1 -10186.609,E2 -10186.609} C_VEL
LIN {X 0,Y 417.545,Z 445.952,A -85,B 0,C 180,E1 -10187.119,E2 -10187.119} C_VEL
LIN {X 0,Y 417.883,Z 437.01,A -85,B 0,C 180,E1 -10190.685,E2 -10190.685} C_VEL
LIN {X 0,Y 418.311,Z 428.107,A -85,B 0,C 180,E1 -10194.31,E2 -10194.31} C_VEL
LIN {X 0,Y 418.781,Z 420.348,A -85,B 0,C 180,E1 -10197.55,E2 -10197.55} C_VEL
LIN {X 0,Y 419.373,Z 412.875,A -85,B 0,C 180,E1 -10200.742,E2 -10200.742} C_VEL
LIN {X 0,Y 420.017,Z 405.294,A -85,B 0,C 180,E1 -10204.096,E2 -10204.096} C_VEL
LIN {X 0,Y 420.286,Z 401.495,A -85,B 0,C 180,E1 -10205.825,E2 -10205.825} C_VEL
LIN {X 0,Y 419.733,Z 396.796,A -85,B 0,C 180,E1 -10208.096,E2 -10208.096} C_VEL
LIN {X 0,Y 418.778,Z 391.168,A -85,B 0,C 180,E1 -10210.956,E2 -10210.956} C_VEL
LIN {X 0,Y 418.277,Z 388.384,A -85,B 0,C 180,E1 -10212.45,E2 -10212.45} C_VEL
LIN {X 0,Y 418.248,Z 388.385,A -85,B 0,C 180,E1 -10215.109,E2 -10215.109} C_VEL
LIN {X 0,Y 418.237,Z 388.388,A -85,B 0,C 180,E1 -10217.766,E2 -10217.766} C_VEL
LIN {X 0,Y 418.251,Z 388.387,A -85,B 0,C 180,E1 -10221.557,E2 -10221.557} C_VEL
LIN {X 0,Y 418.264,Z 388.387,A -85,B 0,C 180,E1 -10225.159,E2 -10225.159} C_VEL
LIN {X 0,Y 418.257,Z 388.387,A -85,B 0,C 180,E1 -10227.472,E2 -10227.472} C_VEL
LIN {X 0,Y 418.277,Z 388.386,A -85,B 0,C 180,E1 -10230.897,E2 -10230.897} C_VEL
LIN {X 0,Y 418.247,Z 388.384,A -85,B 0,C 180,E1 -10234.094,E2 -10234.094} C_VEL
LIN {X 0,Y 418.245,Z 388.389,A -85,B 0,C 180,E1 -10237.263,E2 -10237.263} C_VEL
LIN {X 0,Y 418.297,Z 388.38,A -85,B 0,C 180,E1 -10240.364,E2 -10240.364} C_VEL
LIN {X 0,Y 418.33,Z 388.377,A -85,B 0,C 180,E1 -10243.404,E2 -10243.404} C_VEL
LIN {X 0,Y 418.36,Z 388.375,A -85,B 0,C 180,E1 -10247,E2 -10247} C_VEL
LIN {X 0,Y 418.349,Z 388.373,A -85,B 0,C 180,E1 -10250.328,E2 -10250.328} C_VEL
LIN {X 0,Y 418.48,Z 388.36,A -85,B 0,C 180,E1 -10253.248,E2 -10253.248} C_VEL
LIN {X 0,Y 418.342,Z 388.376,A -85,B 0,C 180,E1 -10255.181,E2 -10255.181} C_VEL
LIN {X 0,Y 418.552,Z 388.347,A -85,B 0,C 180,E1 -10258.075,E2 -10258.075} C_VEL
LIN {X 0,Y 418.677,Z 388.332,A -85,B 0,C 180,E1 -10259.999,E2 -10259.999} C_VEL
LIN {X 0,Y 418.5,Z 388.358,A -85,B 0,C 180,E1 -10262.887,E2 -10262.887} C_VEL
LIN {X 0,Y 418.453,Z 388.361,A -85,B 0,C 180,E1 -10266.563,E2 -10266.563} C_VEL
LIN {X 0,Y 418.346,Z 388.373,A -85,B 0,C 180,E1 -10269.67,E2 -10269.67} C_VEL
LIN {X 0,Y 418.357,Z 388.374,A -85,B 0,C 180,E1 -10272.999,E2 -10272.999} C_VEL
LIN {X 0,Y 418.322,Z 388.379,A -85,B 0,C 180,E1 -10276.733,E2 -10276.733} C_VEL
LIN {X 0,Y 418.28,Z 388.381,A -85,B 0,C 180,E1 -10279.788,E2 -10279.788} C_VEL
LIN {X 0,Y 418.241,Z 388.39,A -85,B 0,C 180,E1 -10282.735,E2 -10282.735} C_VEL
LIN {X 0,Y 418.27,Z 388.383,A -85,B 0,C 180,E1 -10285.903,E2 -10285.903} C_VEL
LIN {X 0,Y 418.276,Z 388.384,A -85,B 0,C 180,E1 -10289.102,E2 -10289.102} C_VEL
LIN {X 0,Y 418.265,Z 388.385,A -85,B 0,C 180,E1 -10292.842,E2 -10292.842} C_VEL
LIN {X 0,Y 418.25,Z 388.387,A -85,B 0,C 180,E1 -10296.235,E2 -10296.235} C_VEL
LIN {X 0,Y 418.24,Z 388.386,A -85,B 0,C 180,E1 -10299.682,E2 -10299.682} C_VEL
LIN {X 0,Y 418.229,Z 388.39,A -85,B 0,C 180,E1 -10302.318,E2 -10302.318} C_VEL
LIN {X 0,Y 418.241,Z 388.388,A -85,B 0,C 180,E1 -10305.106,E2 -10305.106} C_VEL
LIN {X 0,Y 418.239,Z 388.387,A -85,B 0,C 180,E1 -10307.764,E2 -10307.764} C_VEL
LIN {X 0,Y 418.246,Z 388.388,A -85,B 0,C 180,E1 -10310.619,E2 -10310.619} C_VEL
LIN {X 0,Y 418.247,Z 388.387,A -85,B 0,C 180,E1 -10313.973,E2 -10313.973} C_VEL
LIN {X 0,Y 418.261,Z 388.384,A -85,B 0,C 180,E1 -10317.153,E2 -10317.153} C_VEL
LIN {X 0,Y 418.271,Z 388.383,A -85,B 0,C 180,E1 -10320.893,E2 -10320.893} C_VEL
LIN {X 0,Y 418.272,Z 388.384,A -85,B 0,C 180,E1 -10324.093,E2 -10324.093} C_VEL
LIN {X 0,Y 418.239,Z 388.387,A -85,B 0,C 180,E1 -10327.261,E2 -10327.261} C_VEL
LIN {X 0,Y 418.283,Z 388.384,A -85,B 0,C 180,E1 -10330.361,E2 -10330.361} C_VEL
LIN {X 0,Y 418.316,Z 388.376,A -85,B 0,C 180,E1 -10333.401,E2 -10333.401} C_VEL
LIN {X 0,Y 418.344,Z 388.373,A -85,B 0,C 180,E1 -10336.996,E2 -10336.996} C_VEL
LIN {X 0,Y 418.338,Z 388.378,A -85,B 0,C 180,E1 -10340.325,E2 -10340.325} C_VEL
LIN {X 0,Y 418.483,Z 388.356,A -85,B 0,C 180,E1 -10343.245,E2 -10343.245} C_VEL
LIN {X 0,Y 418.331,Z 388.374,A -85,B 0,C 180,E1 -10345.178,E2 -10345.178} C_VEL
LIN {X 0,Y 418.537,Z 388.352,A -85,B 0,C 180,E1 -10348.072,E2 -10348.072} C_VEL
LIN {X 0,Y 418.663,Z 388.337,A -85,B 0,C 180,E1 -10349.996,E2 -10349.996} C_VEL
LIN {X 0,Y 418.501,Z 388.354,A -85,B 0,C 180,E1 -10352.884,E2 -10352.884} C_VEL
LIN {X 0,Y 418.484,Z 388.357,A -85,B 0,C 180,E1 -10356.747,E2 -10356.747} C_VEL
LIN {X 0,Y 418.349,Z 388.375,A -85,B 0,C 180,E1 -10359.667,E2 -10359.667} C_VEL
LIN {X 0,Y 418.321,Z 388.377,A -85,B 0,C 180,E1 -10363.313,E2 -10363.313} C_VEL
LIN {X 0,Y 417.628,Z 388.466,A -85,B 0,C 180,E1 -10364.117,E2 -10364.117} C_VEL
LIN {X 0,Y 414.749,Z 388.822,A -85,B 0,C 180,E1 -10365.422,E2 -10365.422} C_VEL
LIN {X 0,Y 412.331,Z 389.124,A -85,B 0,C 180,E1 -10366.476,E2 -10366.476} C_VEL
LIN {X 0,Y 411.304,Z 389.25,A -85,B 0,C 180,E1 -10367.291,E2 -10367.291} C_VEL
LIN {X 0,Y 411.226,Z 389.26,A -85,B 0,C 180,E1 -10367.567,E2 -10367.567} C_VEL
LIN {X 0,Y 411.179,Z 389.265,A -85,B 0,C 180,E1 -10371.03,E2 -10371.03} C_VEL
LIN {X 0,Y 411.2,Z 389.266,A -85,B 0,C 180,E1 -10374.212,E2 -10374.212} C_VEL
LIN {X 0,Y 411.062,Z 389.283,A -85,B 0,C 180,E1 -10377.487,E2 -10377.487} C_VEL
LIN {X 0,Y 410.662,Z 389.336,A -85,B 0,C 180,E1 -10380.886,E2 -10380.886} C_VEL
LIN {X 0,Y 410.461,Z 389.361,A -85,B 0,C 180,E1 -10382.053,E2 -10382.053} C_VEL
LIN {X 0,Y 410.375,Z 391.799,A -85,B 0,C 180,E1 -10384.713,E2 -10384.713} C_VEL
LIN {X 0,Y 410.318,Z 395.176,A -85,B 0,C 180,E1 -10388.063,E2 -10388.063} C_VEL
LIN {X 0,Y 410.251,Z 398.259,A -85,B 0,C 180,E1 -10391.084,E2 -10391.084} C_VEL
LIN {X 0,Y 410.188,Z 402.122,A -85,B 0,C 180,E1 -10394.752,E2 -10394.752} C_VEL
LIN {X 0,Y 413.369,Z 415.485,A -85,B 0,C 180,E1 -10395.359,E2 -10395.359} C_VEL
LIN {X 0,Y 415.077,Z 423.834,A -85,B 0,C 180,E1 -10395.835,E2 -10395.835} C_VEL
LIN {X 0,Y 414.475,Z 436.568,A -85,B 0,C 180,E1 -10396.626,E2 -10396.626} C_VEL
LIN {X 0,Y 413.831,Z 447.992,A -85,B 0,C 180,E1 -10397.542,E2 -10397.542} C_VEL
LIN {X 0,Y 413.138,Z 457.908,A -85,B 0,C 180,E1 -10398.533,E2 -10398.533} C_VEL
LIN {X 0,Y 412.507,Z 467.08,A -85,B 0,C 180,E1 -10399.654,E2 -10399.654} C_VEL
LIN {X 0,Y 411.824,Z 476.725,A -85,B 0,C 180,E1 -10401.105,E2 -10401.105} C_VEL
LIN {X 0,Y 411.231,Z 484.932,A -85,B 0,C 180,E1 -10402.65,E2 -10402.65} C_VEL
LIN {X 0,Y 410.865,Z 490.532,A -85,B 0,C 180,E1 -10403.954,E2 -10403.954} C_VEL
LIN {X 0,Y 410.487,Z 496.127,A -85,B 0,C 180,E1 -10405.599,E2 -10405.599} C_VEL
LIN {X 0,Y 410.319,Z 499.915,A -85,B 0,C 180,E1 -10407.055,E2 -10407.055} C_VEL
LIN {X 0,Y 410.222,Z 501.692,A -85,B 0,C 180,E1 -10407.922,E2 -10407.922} C_VEL
LIN {X 0,Y 410.025,Z 503.539,A -85,B 0,C 180,E1 -10409.056,E2 -10409.056} C_VEL
LIN {X 0,Y 409.946,Z 505.31,A -85,B 0,C 180,E1 -10410.955,E2 -10410.955} C_VEL
LIN {X 0,Y 409.929,Z 505.567,A -85,B 0,C 180,E1 -10413.052,E2 -10413.052} C_VEL
LIN {X 0,Y 410.029,Z 504.54,A -85,B 0,C 180,E1 -10414.628,E2 -10414.628} C_VEL
LIN {X 0,Y 410.175,Z 503.2,A -85,B 0,C 180,E1 -10415.72,E2 -10415.72} C_VEL
LIN {X 0,Y 410.342,Z 501.402,A -85,B 0,C 180,E1 -10416.802,E2 -10416.802} C_VEL
LIN {X 0,Y 410.618,Z 497.701,A -85,B 0,C 180,E1 -10418.41,E2 -10418.41} C_VEL
LIN {X 0,Y 411.009,Z 492.346,A -85,B 0,C 180,E1 -10420.114,E2 -10420.114} C_VEL
LIN {X 0,Y 411.459,Z 486.435,A -85,B 0,C 180,E1 -10421.58,E2 -10421.58} C_VEL
LIN {X 0,Y 412.175,Z 478.479,A -85,B 0,C 180,E1 -10423.151,E2 -10423.151} C_VEL
LIN {X 0,Y 412.843,Z 470.285,A -85,B 0,C 180,E1 -10424.449,E2 -10424.449} C_VEL
LIN {X 0,Y 413.635,Z 460.028,A -85,B 0,C 180,E1 -10425.768,E2 -10425.768} C_VEL
LIN {X 0,Y 414.384,Z 450.448,A -85,B 0,C 180,E1 -10426.765,E2 -10426.765} C_VEL
LIN {X 0,Y 415.073,Z 439.915,A -85,B 0,C 180,E1 -10427.658,E2 -10427.658} C_VEL
LIN {X 0,Y 415.768,Z 428.149,A -85,B 0,C 180,E1 -10428.439,E2 -10428.439} C_VEL
LIN {X 0,Y 415.793,Z 424.369,A -85,B 0,C 180,E1 -10428.66,E2 -10428.66} C_VEL
LIN {X 0,Y 413.059,Z 412.837,A -85,B 0,C 180,E1 -10429.353,E2 -10429.353} C_VEL
LIN {X 0,Y 410.504,Z 404.235,A -85,B 0,C 180,E1 -10429.801,E2 -10429.801} C_VEL
LIN {X 0,Y 410.699,Z 401.202,A -85,B 0,C 180,E1 -10433.121,E2 -10433.121} C_VEL
LIN {X 0,Y 410.888,Z 399.415,A -85,B 0,C 180,E1 -10435.095,E2 -10435.095} C_VEL
LIN {X 0,Y 411.108,Z 395.205,A -85,B 0,C 180,E1 -10440.001,E2 -10440.001} C_VEL
LIN {X 0,Y 411.277,Z 394.376,A -85,B 0,C 180,E1 -10440.98,E2 -10440.98} C_VEL
LIN {X 0,Y 411.398,Z 390.449,A -85,B 0,C 180,E1 -10445.884,E2 -10445.884} C_VEL
LIN {X 0,Y 411.351,Z 389.251,A -85,B 0,C 180,E1 -10447.857,E2 -10447.857} C_VEL
LIN {X 0,Y 411.281,Z 389.256,A -85,B 0,C 180,E1 -10450.835,E2 -10450.835} C_VEL
LIN {X 0,Y 411.232,Z 389.262,A -85,B 0,C 180,E1 -10453.844,E2 -10453.844} C_VEL
LIN {X 0,Y 411.268,Z 389.256,A -85,B 0,C 180,E1 -10456.889,E2 -10456.889} C_VEL
LIN {X 0,Y 411.223,Z 389.263,A -85,B 0,C 180,E1 -10459.988,E2 -10459.988} C_VEL
LIN {X 0,Y 411.199,Z 389.264,A -85,B 0,C 180,E1 -10463.149,E2 -10463.149} C_VEL
LIN {X 0,Y 411.21,Z 389.263,A -85,B 0,C 180,E1 -10466.384,E2 -10466.384} C_VEL
LIN {X 0,Y 411.181,Z 389.267,A -85,B 0,C 180,E1 -10469.715,E2 -10469.715} C_VEL
LIN {X 0,Y 411.179,Z 389.268,A -85,B 0,C 180,E1 -10473.159,E2 -10473.159} C_VEL
LIN {X 0,Y 411.17,Z 389.27,A -85,B 0,C 180,E1 -10476.557,E2 -10476.557} C_VEL
LIN {X 0,Y 411.206,Z 389.266,A -85,B 0,C 180,E1 -10479.734,E2 -10479.734} C_VEL
LIN {X 0,Y 411.202,Z 389.267,A -85,B 0,C 180,E1 -10483.131,E2 -10483.131} C_VEL
